(* Visualisation VISU_2_UDP
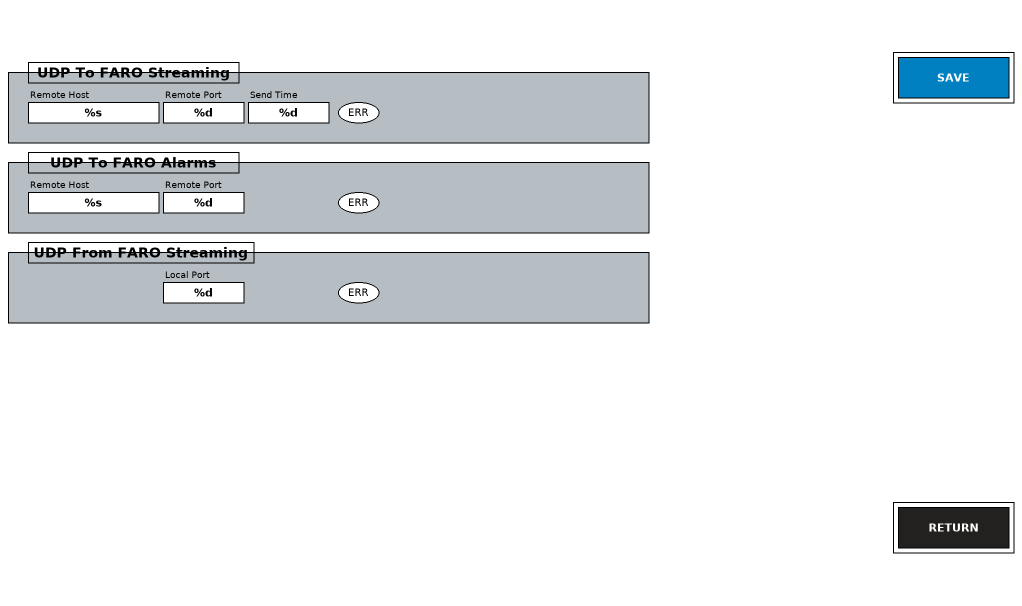
rounded rectangle at (905,505)-(1016,546): text "RETURN"; opens VISU_1_ALARMS
rectangle at (20,0)-(506,51): text "UDP STREAMING"
rectangle at (20,550)-(351,601): text "%s"; shows INPUTS.sVisuTime
rounded rectangle at (905,55)-(1016,96): text "SAVE"; alarm colour if PARAMS.Save; toggles PARAMS.Save
rectangle at (35,100)-(166,121): text "%s"; shows PARAMS.sUDPSendHost; editable
ellipse at (345,100)-(386,121): text "ERR"; alarm colour if TOFARO.fbUdpSend.bError
rectangle at (170,100)-(251,121): text "%d"; shows PARAMS.nUDPSendPort; editable
rectangle at (255,100)-(336,121): text "%d"; shows PARAMS.nUDPSendTime; editable 0..
rectangle at (35,85)-(126,101): text "Remote Host"
rectangle at (170,85)-(251,101): text "Remote Port"
rectangle at (255,85)-(336,101): text "Send Time"
rectangle at (35,60)-(246,81): text "UDP To FARO Streaming"
rectangle at (730,550)-(896,601): text "SAVED!"; invisible if PARAMS.Saved
ellipse at (345,280)-(386,301): text "ERR"; alarm colour if TOFARO.fbUdpRecv.bError
rectangle at (170,280)-(251,301): text "%d"; shows PARAMS.nUDPRecvPort; editable
rectangle at (170,265)-(251,281): text "Local Port"
rectangle at (35,240)-(261,261): text "UDP From FARO Streaming"
rectangle at (35,190)-(166,211): text "%s"; shows PARAMS.sUDPAlarmsHost; editable
ellipse at (345,190)-(386,211): text "ERR"; alarm colour if ALARMS.fbUdpSend.bError
rectangle at (170,190)-(251,211): text "%d"; shows PARAMS.nUDPAlarmsPort; editable
rectangle at (35,175)-(126,191): text "Remote Host"
rectangle at (170,175)-(251,191): text "Remote Port"
rectangle at (35,150)-(246,171): text "UDP To FARO Alarms"
5 more shapes without text or variables
*)

(* Visualisation VISU_CAL_CYLINDERS1
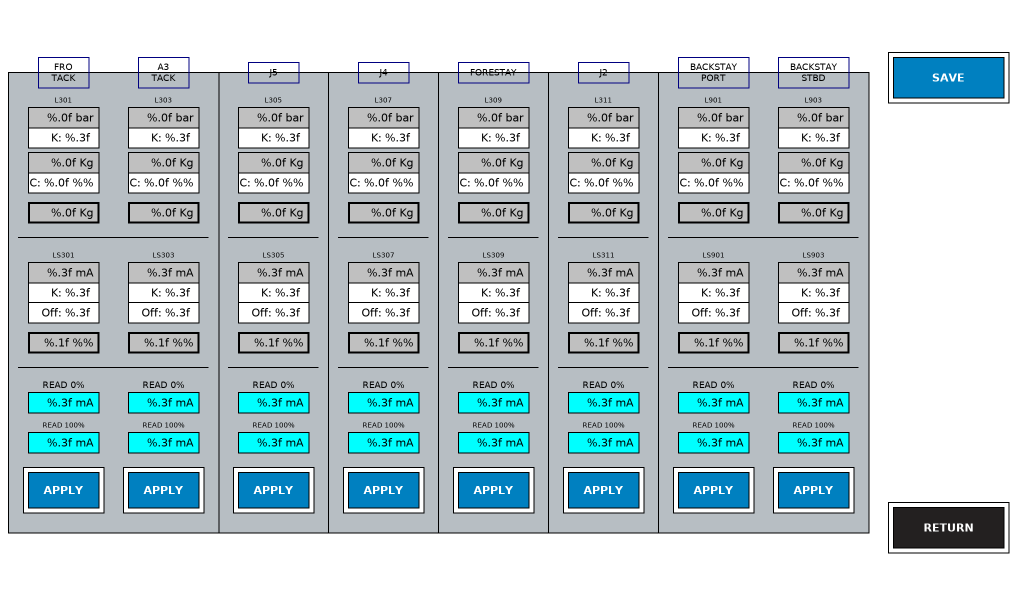
rectangle at (20,0)-(426,51): text "CAL: CYLINDERS 1"
rectangle at (20,550)-(331,601): text "%s"; shows INPUTS.sVisuTime
rounded rectangle at (905,55)-(1016,96): text "SAVE"; alarm colour if PARAMS.Save; toggles PARAMS.Save
rounded rectangle at (905,505)-(1016,546): text "RETURN"; opens VISU_1_CYLINDERS1
rectangle at (725,550)-(891,601): text "SAVED!"; invisible if PARAMS.Saved
rectangle at (40,245)-(111,261): text "LS301"
rectangle at (40,280)-(111,301): text "K: %.3f"; shows LS301.Cal_K; runs INTERN ASSIGN INPUTS.PresSelCalStbd[9]:=(FALSE); editable
rectangle at (40,260)-(111,281): text "%.3f mA"; shows LS301.Raw; alarm colour if LS301.Err; runs INTERN ASSIGN INPUTS.PresSelCalStbd[9]:=(FALSE)
rectangle at (40,300)-(111,321): text "Off: %.3f"; shows LS301.Cal_Off; runs INTERN ASSIGN INPUTS.PresSelCalStbd[9]:=(FALSE); editable
rectangle at (40,430)-(111,451): text "%.3f mA"; shows LS301.Cal_Max; alarm colour if LS301.Cal_Max = 0.0; runs INTERN ASSIGN INPUTS.PresSelCalStbd[9]:=(FALSE); editable
rectangle at (40,375)-(111,391): text "READ 0%"
rectangle at (40,415)-(111,431): text "READ 100%"
rounded rectangle at (40,470)-(111,506): text "APPLY"; toggles LS301.Cal_Apply
rectangle at (140,245)-(211,261): text "LS303"
rectangle at (140,280)-(211,301): text "K: %.3f"; shows LS303.Cal_K; runs INTERN ASSIGN INPUTS.PresSelCalStbd[9]:=(FALSE); editable
rectangle at (140,260)-(211,281): text "%.3f mA"; shows LS303.Raw; alarm colour if LS303.Err; runs INTERN ASSIGN INPUTS.PresSelCalStbd[9]:=(FALSE)
rectangle at (140,300)-(211,321): text "Off: %.3f"; shows LS303.Cal_Off; runs INTERN ASSIGN INPUTS.PresSelCalStbd[9]:=(FALSE); editable
rectangle at (140,430)-(211,451): text "%.3f mA"; shows LS303.Cal_Max; alarm colour if LS303.Cal_Max = 0.0; runs INTERN ASSIGN INPUTS.PresSelCalStbd[9]:=(FALSE); editable
rounded rectangle at (140,470)-(211,506): text "APPLY"; toggles LS303.Cal_Apply
rectangle at (690,280)-(761,301): text "K: %.3f"; shows LS901.Cal_K; runs INTERN ASSIGN INPUTS.PresSelCalStbd[9]:=(FALSE); editable
rectangle at (690,260)-(761,281): text "%.3f mA"; shows LS901.Raw; alarm colour if LS901.Err; runs INTERN ASSIGN INPUTS.PresSelCalStbd[9]:=(FALSE)
rectangle at (690,300)-(761,321): text "Off: %.3f"; shows LS901.Cal_Off; runs INTERN ASSIGN INPUTS.PresSelCalStbd[9]:=(FALSE); editable
rectangle at (690,390)-(761,411): text "%.3f mA"; shows LS901.Cal_Min; alarm colour if LS901.Cal_Min = 0.0; runs INTERN ASSIGN INPUTS.PresSelCalStbd[9]:=(FALSE); editable
rectangle at (690,430)-(761,451): text "%.3f mA"; shows LS901.Cal_Max; alarm colour if LS901.Cal_Max = 0.0; runs INTERN ASSIGN INPUTS.PresSelCalStbd[9]:=(FALSE); editable
rounded rectangle at (690,470)-(761,506): text "APPLY"; toggles LS901.Cal_Apply
rectangle at (790,280)-(861,301): text "K: %.3f"; shows LS903.Cal_K; runs INTERN ASSIGN INPUTS.PresSelCalStbd[9]:=(FALSE); editable
rectangle at (790,260)-(861,281): text "%.3f mA"; shows LS903.Raw; alarm colour if LS903.Err; runs INTERN ASSIGN INPUTS.PresSelCalStbd[9]:=(FALSE)
rectangle at (790,300)-(861,321): text "Off: %.3f"; shows LS903.Cal_Off; runs INTERN ASSIGN INPUTS.PresSelCalStbd[9]:=(FALSE); editable
rectangle at (790,390)-(861,411): text "%.3f mA"; shows LS903.Cal_Min; alarm colour if LS903.Cal_Min = 0.0; runs INTERN ASSIGN INPUTS.PresSelCalStbd[9]:=(FALSE); editable
rectangle at (790,430)-(861,451): text "%.3f mA"; shows LS903.Cal_Max; alarm colour if LS903.Cal_Max = 0.0; runs INTERN ASSIGN INPUTS.PresSelCalStbd[9]:=(FALSE); editable
rounded rectangle at (790,470)-(861,506): text "APPLY"; toggles LS903.Cal_Apply
rectangle at (580,280)-(651,301): text "K: %.3f"; shows LS311.Cal_K; runs INTERN ASSIGN INPUTS.PresSelCalStbd[9]:=(FALSE); editable
rectangle at (580,260)-(651,281): text "%.3f mA"; shows LS311.Raw; alarm colour if LS311.Err; runs INTERN ASSIGN INPUTS.PresSelCalStbd[9]:=(FALSE)
rectangle at (580,300)-(651,321): text "Off: %.3f"; shows LS311.Cal_Off; runs INTERN ASSIGN INPUTS.PresSelCalStbd[9]:=(FALSE); editable
rectangle at (580,390)-(651,411): text "%.3f mA"; shows LS311.Cal_Min; alarm colour if LS311.Cal_Min = 0.0; runs INTERN ASSIGN INPUTS.PresSelCalStbd[9]:=(FALSE); editable
rectangle at (580,430)-(651,451): text "%.3f mA"; shows LS311.Cal_Max; alarm colour if LS311.Cal_Max = 0.0; runs INTERN ASSIGN INPUTS.PresSelCalStbd[9]:=(FALSE); editable
rounded rectangle at (580,470)-(651,506): text "APPLY"; toggles LS311.Cal_Apply
rectangle at (250,280)-(321,301): text "K: %.3f"; shows LS305.Cal_K; runs INTERN ASSIGN INPUTS.PresSelCalStbd[9]:=(FALSE); editable
rectangle at (250,260)-(321,281): text "%.3f mA"; shows LS305.Raw; alarm colour if LS305.Err; runs INTERN ASSIGN INPUTS.PresSelCalStbd[9]:=(FALSE)
rectangle at (250,300)-(321,321): text "Off: %.3f"; shows LS305.Cal_Off; runs INTERN ASSIGN INPUTS.PresSelCalStbd[9]:=(FALSE); editable
rectangle at (250,390)-(321,411): text "%.3f mA"; shows LS305.Cal_Min; alarm colour if LS305.Cal_Min = 0.0; runs INTERN ASSIGN INPUTS.PresSelCalStbd[9]:=(FALSE); editable
rectangle at (250,430)-(321,451): text "%.3f mA"; shows LS305.Cal_Max; alarm colour if LS305.Cal_Max = 0.0; runs INTERN ASSIGN INPUTS.PresSelCalStbd[9]:=(FALSE); editable
rounded rectangle at (250,470)-(321,506): text "APPLY"; toggles LS305.Cal_Apply
rectangle at (360,280)-(431,301): text "K: %.3f"; shows LS307.Cal_K; runs INTERN ASSIGN INPUTS.PresSelCalStbd[9]:=(FALSE); editable
rectangle at (360,260)-(431,281): text "%.3f mA"; shows LS307.Raw; alarm colour if LS307.Err; runs INTERN ASSIGN INPUTS.PresSelCalStbd[9]:=(FALSE)
rectangle at (360,300)-(431,321): text "Off: %.3f"; shows LS307.Cal_Off; runs INTERN ASSIGN INPUTS.PresSelCalStbd[9]:=(FALSE); editable
rectangle at (360,390)-(431,411): text "%.3f mA"; shows LS307.Cal_Min; alarm colour if LS307.Cal_Min = 0.0; runs INTERN ASSIGN INPUTS.PresSelCalStbd[9]:=(FALSE); editable
rectangle at (360,430)-(431,451): text "%.3f mA"; shows LS307.Cal_Max; alarm colour if LS307.Cal_Max = 0.0; runs INTERN ASSIGN INPUTS.PresSelCalStbd[9]:=(FALSE); editable
rounded rectangle at (360,470)-(431,506): text "APPLY"; toggles LS307.Cal_Apply
rectangle at (40,390)-(111,411): text "%.3f mA"; shows LS301.Cal_Min; alarm colour if LS301.Cal_Min = 0.0; runs INTERN ASSIGN INPUTS.PresSelCalStbd[9]:=(FALSE); editable
rectangle at (140,390)-(211,411): text "%.3f mA"; shows LS303.Cal_Min; alarm colour if LS303.Cal_Min = 0.0; runs INTERN ASSIGN INPUTS.PresSelCalStbd[9]:=(FALSE); editable
rectangle at (40,90)-(111,106): text "L301"
rectangle at (40,200)-(111,221): text "%.0f Kg"; shows L301.Kg; runs INTERN ASSIGN INPUTS.PresSelCalStbd[9]:=(FALSE)
rectangle at (40,125)-(111,146): text "K: %.3f"; shows L301.Cal_K; runs INTERN ASSIGN INPUTS.PresSelCalStbd[9]:=(FALSE); editable
rectangle at (40,105)-(111,126): text "%.0f bar"; shows P301.Bar; alarm colour if P301.Err; runs INTERN ASSIGN INPUTS.PresSelCalStbd[9]:=(FALSE)
rectangle at (40,170)-(111,191): text "C: %.0f %%"; shows L301.Cal_C; runs INTERN ASSIGN INPUTS.PresSelCalStbd[9]:=(FALSE); editable
rectangle at (40,150)-(111,171): text "%.0f Kg"; shows L301.Raw; runs INTERN ASSIGN INPUTS.PresSelCalStbd[9]:=(FALSE)
rectangle at (40,330)-(111,351): text "%.1f %%"; shows LS301.Pos; runs INTERN ASSIGN INPUTS.PresSelCalStbd[9]:=(FALSE)
rectangle at (140,330)-(211,351): text "%.1f %%"; shows LS303.Pos; runs INTERN ASSIGN INPUTS.PresSelCalStbd[9]:=(FALSE)
rectangle at (690,330)-(761,351): text "%.1f %%"; shows LS901.Pos; runs INTERN ASSIGN INPUTS.PresSelCalStbd[9]:=(FALSE)
rectangle at (790,330)-(861,351): text "%.1f %%"; shows LS903.Pos; runs INTERN ASSIGN INPUTS.PresSelCalStbd[9]:=(FALSE)
rectangle at (580,330)-(651,351): text "%.1f %%"; shows LS311.Pos; runs INTERN ASSIGN INPUTS.PresSelCalStbd[9]:=(FALSE)
rectangle at (250,330)-(321,351): text "%.1f %%"; shows LS305.Pos; runs INTERN ASSIGN INPUTS.PresSelCalStbd[9]:=(FALSE)
rectangle at (360,330)-(431,351): text "%.1f %%"; shows LS307.Pos; runs INTERN ASSIGN INPUTS.PresSelCalStbd[9]:=(FALSE)
rectangle at (470,280)-(541,301): text "K: %.3f"; shows LS309.Cal_K; runs INTERN ASSIGN INPUTS.PresSelCalStbd[9]:=(FALSE); editable
rectangle at (470,260)-(541,281): text "%.3f mA"; shows LS309.Raw; alarm colour if LS309.Err; runs INTERN ASSIGN INPUTS.PresSelCalStbd[9]:=(FALSE)
rectangle at (470,300)-(541,321): text "Off: %.3f"; shows LS309.Cal_Off; runs INTERN ASSIGN INPUTS.PresSelCalStbd[9]:=(FALSE); editable
rectangle at (470,390)-(541,411): text "%.3f mA"; shows LS309.Cal_Min; alarm colour if LS309.Cal_Min = 0.0; runs INTERN ASSIGN INPUTS.PresSelCalStbd[9]:=(FALSE); editable
rectangle at (470,430)-(541,451): text "%.3f mA"; shows LS309.Cal_Max; alarm colour if LS309.Cal_Max = 0.0; runs INTERN ASSIGN INPUTS.PresSelCalStbd[9]:=(FALSE); editable
rounded rectangle at (470,470)-(541,506): text "APPLY"; toggles LS309.Cal_Apply
rectangle at (470,330)-(541,351): text "%.1f %%"; shows LS309.Pos; runs INTERN ASSIGN INPUTS.PresSelCalStbd[9]:=(FALSE)
rectangle at (140,90)-(211,106): text "L303"
rectangle at (140,200)-(211,221): text "%.0f Kg"; shows L303.Kg; runs INTERN ASSIGN INPUTS.PresSelCalStbd[9]:=(FALSE)
rectangle at (140,125)-(211,146): text "K: %.3f"; shows L303.Cal_K; runs INTERN ASSIGN INPUTS.PresSelCalStbd[9]:=(FALSE); editable
rectangle at (140,105)-(211,126): text "%.0f bar"; shows P303.Bar; alarm colour if P303.Err; runs INTERN ASSIGN INPUTS.PresSelCalStbd[9]:=(FALSE)
rectangle at (140,170)-(211,191): text "C: %.0f %%"; shows L303.Cal_C; runs INTERN ASSIGN INPUTS.PresSelCalStbd[9]:=(FALSE); editable
rectangle at (140,150)-(211,171): text "%.0f Kg"; shows L303.Raw; runs INTERN ASSIGN INPUTS.PresSelCalStbd[9]:=(FALSE)
rectangle at (250,90)-(321,106): text "L305"
rectangle at (250,200)-(321,221): text "%.0f Kg"; shows L305.Kg; runs INTERN ASSIGN INPUTS.PresSelCalStbd[9]:=(FALSE)
rectangle at (250,125)-(321,146): text "K: %.3f"; shows L305.Cal_K; runs INTERN ASSIGN INPUTS.PresSelCalStbd[9]:=(FALSE); editable
rectangle at (250,105)-(321,126): text "%.0f bar"; shows P305.Bar; alarm colour if P305.Err; runs INTERN ASSIGN INPUTS.PresSelCalStbd[9]:=(FALSE)
rectangle at (250,170)-(321,191): text "C: %.0f %%"; shows L305.Cal_C; runs INTERN ASSIGN INPUTS.PresSelCalStbd[9]:=(FALSE); editable
rectangle at (250,150)-(321,171): text "%.0f Kg"; shows L305.Raw; runs INTERN ASSIGN INPUTS.PresSelCalStbd[9]:=(FALSE)
rectangle at (250,245)-(321,261): text "LS305"
rectangle at (360,245)-(431,261): text "LS307"
rectangle at (470,245)-(541,261): text "LS309"
rectangle at (580,245)-(651,261): text "LS311"
rectangle at (690,245)-(761,261): text "LS901"
rectangle at (790,245)-(861,261): text "LS903"
rectangle at (360,90)-(431,106): text "L307"
rectangle at (360,200)-(431,221): text "%.0f Kg"; shows L307.Kg; runs INTERN ASSIGN INPUTS.PresSelCalStbd[9]:=(FALSE)
rectangle at (360,125)-(431,146): text "K: %.3f"; shows L307.Cal_K; runs INTERN ASSIGN INPUTS.PresSelCalStbd[9]:=(FALSE); editable
rectangle at (360,105)-(431,126): text "%.0f bar"; shows P307.Bar; alarm colour if P307.Err; runs INTERN ASSIGN INPUTS.PresSelCalStbd[9]:=(FALSE)
rectangle at (360,170)-(431,191): text "C: %.0f %%"; shows L307.Cal_C; runs INTERN ASSIGN INPUTS.PresSelCalStbd[9]:=(FALSE); editable
rectangle at (360,150)-(431,171): text "%.0f Kg"; shows L307.Raw; runs INTERN ASSIGN INPUTS.PresSelCalStbd[9]:=(FALSE)
rectangle at (470,90)-(541,106): text "L309"
rectangle at (470,200)-(541,221): text "%.0f Kg"; shows L309.Kg; runs INTERN ASSIGN INPUTS.PresSelCalStbd[9]:=(FALSE)
rectangle at (470,125)-(541,146): text "K: %.3f"; shows L309.Cal_K; runs INTERN ASSIGN INPUTS.PresSelCalStbd[9]:=(FALSE); editable
rectangle at (470,105)-(541,126): text "%.0f bar"; shows P309.Bar; alarm colour if P309.Err; runs INTERN ASSIGN INPUTS.PresSelCalStbd[9]:=(FALSE)
rectangle at (470,170)-(541,191): text "C: %.0f %%"; shows L309.Cal_C; runs INTERN ASSIGN INPUTS.PresSelCalStbd[9]:=(FALSE); editable
rectangle at (470,150)-(541,171): text "%.0f Kg"; shows L309.Raw; runs INTERN ASSIGN INPUTS.PresSelCalStbd[9]:=(FALSE)
rectangle at (580,90)-(651,106): text "L311"
rectangle at (580,200)-(651,221): text "%.0f Kg"; shows L311.Kg; runs INTERN ASSIGN INPUTS.PresSelCalStbd[9]:=(FALSE)
rectangle at (580,125)-(651,146): text "K: %.3f"; shows L311.Cal_K; runs INTERN ASSIGN INPUTS.PresSelCalStbd[9]:=(FALSE); editable
rectangle at (580,105)-(651,126): text "%.0f bar"; shows P311.Bar; alarm colour if P311.Err; runs INTERN ASSIGN INPUTS.PresSelCalStbd[9]:=(FALSE)
rectangle at (580,170)-(651,191): text "C: %.0f %%"; shows L311.Cal_C; runs INTERN ASSIGN INPUTS.PresSelCalStbd[9]:=(FALSE); editable
rectangle at (580,150)-(651,171): text "%.0f Kg"; shows L311.Raw; runs INTERN ASSIGN INPUTS.PresSelCalStbd[9]:=(FALSE)
rectangle at (690,90)-(761,106): text "L901"
rectangle at (690,200)-(761,221): text "%.0f Kg"; shows L901.Kg; runs INTERN ASSIGN INPUTS.PresSelCalStbd[9]:=(FALSE)
rectangle at (690,125)-(761,146): text "K: %.3f"; shows L901.Cal_K; runs INTERN ASSIGN INPUTS.PresSelCalStbd[9]:=(FALSE); editable
rectangle at (690,105)-(761,126): text "%.0f bar"; shows P901.Bar; alarm colour if P901.Err; runs INTERN ASSIGN INPUTS.PresSelCalStbd[9]:=(FALSE)
rectangle at (690,170)-(761,191): text "C: %.0f %%"; shows L901.Cal_C; runs INTERN ASSIGN INPUTS.PresSelCalStbd[9]:=(FALSE); editable
rectangle at (690,150)-(761,171): text "%.0f Kg"; shows L901.Raw; runs INTERN ASSIGN INPUTS.PresSelCalStbd[9]:=(FALSE)
rectangle at (790,90)-(861,106): text "L903"
rectangle at (790,200)-(861,221): text "%.0f Kg"; shows L903.Kg; runs INTERN ASSIGN INPUTS.PresSelCalStbd[9]:=(FALSE)
rectangle at (790,125)-(861,146): text "K: %.3f"; shows L903.Cal_K; runs INTERN ASSIGN INPUTS.PresSelCalStbd[9]:=(FALSE); editable
rectangle at (790,105)-(861,126): text "%.0f bar"; shows P903.Bar; alarm colour if P903.Err; runs INTERN ASSIGN INPUTS.PresSelCalStbd[9]:=(FALSE)
rectangle at (790,170)-(861,191): text "C: %.0f %%"; shows L903.Cal_C; runs INTERN ASSIGN INPUTS.PresSelCalStbd[9]:=(FALSE); editable
rectangle at (790,150)-(861,171): text "%.0f Kg"; shows L903.Raw; runs INTERN ASSIGN INPUTS.PresSelCalStbd[9]:=(FALSE)
rectangle at (260,60)-(311,81): text "J5"
rectangle at (370,60)-(421,81): text "J4"
rectangle at (470,60)-(541,81): text "FORESTAY"
rectangle at (590,60)-(641,81): text "J2"
rectangle at (690,55)-(761,86): text "BACKSTAY / PORT"
rectangle at (790,55)-(861,86): text "BACKSTAY / STBD"
rectangle at (150,55)-(201,86): text "A3 / TACK"
rectangle at (50,55)-(101,86): text "FRO / TACK"
rectangle at (140,375)-(211,391): text "READ 0%"
rectangle at (140,415)-(211,431): text "READ 100%"
rectangle at (250,375)-(321,391): text "READ 0%"
rectangle at (250,415)-(321,431): text "READ 100%"
rectangle at (360,375)-(431,391): text "READ 0%"
rectangle at (360,415)-(431,431): text "READ 100%"
rectangle at (470,375)-(541,391): text "READ 0%"
rectangle at (470,415)-(541,431): text "READ 100%"
rectangle at (580,375)-(651,391): text "READ 0%"
rectangle at (580,415)-(651,431): text "READ 100%"
rectangle at (690,375)-(761,391): text "READ 0%"
rectangle at (690,415)-(761,431): text "READ 100%"
rectangle at (790,375)-(861,391): text "READ 0%"
rectangle at (790,415)-(861,431): text "READ 100%"
28 more shapes without text or variables
*)

(* Visualisation VISU_CAL_CYLINDERS2
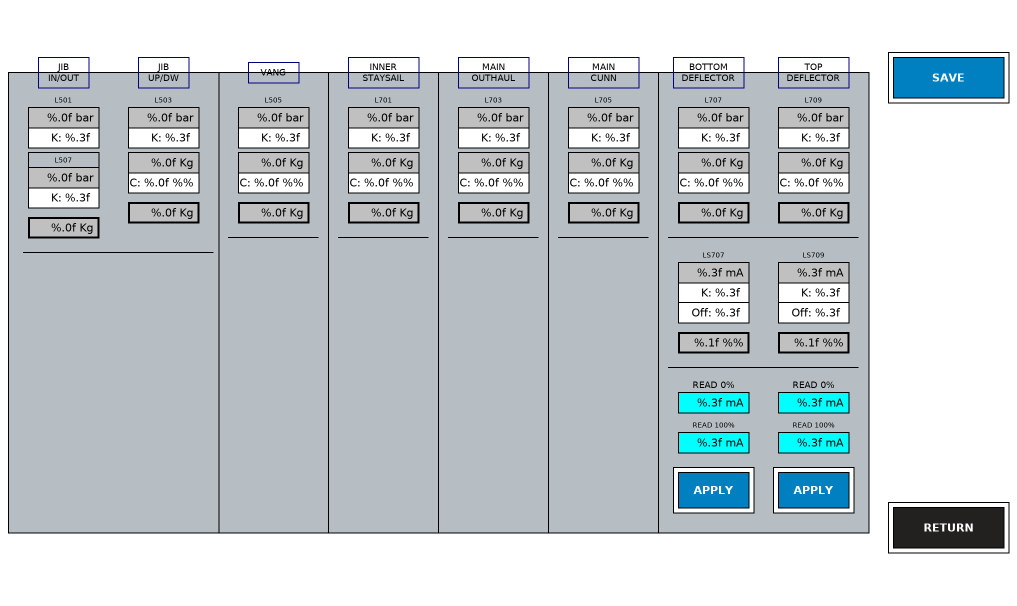
rectangle at (20,0)-(426,51): text "CAL: CYLINDERS 2"
rectangle at (20,550)-(331,601): text "%s"; shows INPUTS.sVisuTime
rounded rectangle at (905,55)-(1016,96): text "SAVE"; alarm colour if PARAMS.Save; toggles PARAMS.Save
rounded rectangle at (905,505)-(1016,546): text "RETURN"; opens VISU_1_CYLINDERS2
rectangle at (730,550)-(896,601): text "SAVED!"; invisible if PARAMS.Saved
rectangle at (690,245)-(761,261): text "LS707"
rectangle at (690,280)-(761,301): text "K: %.3f"; shows LS707.Cal_K; runs INTERN ASSIGN INPUTS.PresSelCalStbd[9]:=(FALSE); editable
rectangle at (690,260)-(761,281): text "%.3f mA"; shows LS707.Raw; alarm colour if LS707.Err; runs INTERN ASSIGN INPUTS.PresSelCalStbd[9]:=(FALSE)
rectangle at (690,300)-(761,321): text "Off: %.3f"; shows LS707.Cal_Off; runs INTERN ASSIGN INPUTS.PresSelCalStbd[9]:=(FALSE); editable
rectangle at (690,430)-(761,451): text "%.3f mA"; shows LS707.Cal_Max; alarm colour if LS707.Cal_Max = 0.0; runs INTERN ASSIGN INPUTS.PresSelCalStbd[9]:=(FALSE); editable
rectangle at (690,375)-(761,391): text "READ 0%"
rectangle at (690,415)-(761,431): text "READ 100%"
rounded rectangle at (690,470)-(761,506): text "APPLY"; toggles LS707.Cal_Apply
rectangle at (790,245)-(861,261): text "LS709"
rectangle at (790,280)-(861,301): text "K: %.3f"; shows LS709.Cal_K; runs INTERN ASSIGN INPUTS.PresSelCalStbd[9]:=(FALSE); editable
rectangle at (790,260)-(861,281): text "%.3f mA"; shows LS709.Raw; alarm colour if LS709.Err; runs INTERN ASSIGN INPUTS.PresSelCalStbd[9]:=(FALSE)
rectangle at (790,300)-(861,321): text "Off: %.3f"; shows LS709.Cal_Off; runs INTERN ASSIGN INPUTS.PresSelCalStbd[9]:=(FALSE); editable
rectangle at (790,430)-(861,451): text "%.3f mA"; shows LS709.Cal_Max; alarm colour if LS709.Cal_Max = 0.0; runs INTERN ASSIGN INPUTS.PresSelCalStbd[9]:=(FALSE); editable
rectangle at (790,375)-(861,391): text "READ 0%"
rectangle at (790,415)-(861,431): text "READ 100%"
rounded rectangle at (790,470)-(861,506): text "APPLY"; toggles LS709.Cal_Apply
rectangle at (690,390)-(761,411): text "%.3f mA"; shows LS707.Cal_Min; alarm colour if LS707.Cal_Min = 0.0; runs INTERN ASSIGN INPUTS.PresSelCalStbd[9]:=(FALSE); editable
rectangle at (790,390)-(861,411): text "%.3f mA"; shows LS709.Cal_Min; alarm colour if LS709.Cal_Min = 0.0; runs INTERN ASSIGN INPUTS.PresSelCalStbd[9]:=(FALSE); editable
rectangle at (690,330)-(761,351): text "%.1f %%"; shows LS707.Pos; runs INTERN ASSIGN INPUTS.PresSelCalStbd[9]:=(FALSE)
rectangle at (790,330)-(861,351): text "%.1f %%"; shows LS709.Pos; runs INTERN ASSIGN INPUTS.PresSelCalStbd[9]:=(FALSE)
rectangle at (40,90)-(111,106): text "L501"
rectangle at (40,215)-(111,236): text "%.0f Kg"; shows L501_7; runs INTERN ASSIGN INPUTS.PresSelCalStbd[9]:=(FALSE)
rectangle at (40,125)-(111,146): text "K: %.3f"; shows L501.Cal_K; runs INTERN ASSIGN INPUTS.PresSelCalStbd[9]:=(FALSE); editable
rectangle at (40,105)-(111,126): text "%.0f bar"; shows P501.Bar; alarm colour if P501.Err; runs INTERN ASSIGN INPUTS.PresSelCalStbd[9]:=(FALSE)
rectangle at (140,90)-(211,106): text "L503"
rectangle at (140,200)-(211,221): text "%.0f Kg"; shows L503.Kg; runs INTERN ASSIGN INPUTS.PresSelCalStbd[9]:=(FALSE)
rectangle at (140,125)-(211,146): text "K: %.3f"; shows L503.Cal_K; runs INTERN ASSIGN INPUTS.PresSelCalStbd[9]:=(FALSE); editable
rectangle at (140,105)-(211,126): text "%.0f bar"; shows P503.Bar; alarm colour if P503.Err; runs INTERN ASSIGN INPUTS.PresSelCalStbd[9]:=(FALSE)
rectangle at (140,170)-(211,191): text "C: %.0f %%"; shows L503.Cal_C; runs INTERN ASSIGN INPUTS.PresSelCalStbd[9]:=(FALSE); editable
rectangle at (140,150)-(211,171): text "%.0f Kg"; shows L503.Raw; runs INTERN ASSIGN INPUTS.PresSelCalStbd[9]:=(FALSE)
rectangle at (690,90)-(761,106): text "L707"
rectangle at (690,200)-(761,221): text "%.0f Kg"; shows L707.Kg; runs INTERN ASSIGN INPUTS.PresSelCalStbd[9]:=(FALSE)
rectangle at (690,125)-(761,146): text "K: %.3f"; shows L707.Cal_K; runs INTERN ASSIGN INPUTS.PresSelCalStbd[9]:=(FALSE); editable
rectangle at (690,105)-(761,126): text "%.0f bar"; shows P707.Bar; alarm colour if P707.Err; runs INTERN ASSIGN INPUTS.PresSelCalStbd[9]:=(FALSE)
rectangle at (690,170)-(761,191): text "C: %.0f %%"; shows L707.Cal_C; runs INTERN ASSIGN INPUTS.PresSelCalStbd[9]:=(FALSE); editable
rectangle at (690,150)-(761,171): text "%.0f Kg"; shows L707.Raw; runs INTERN ASSIGN INPUTS.PresSelCalStbd[9]:=(FALSE)
rectangle at (790,90)-(861,106): text "L709"
rectangle at (790,200)-(861,221): text "%.0f Kg"; shows L709.Kg; runs INTERN ASSIGN INPUTS.PresSelCalStbd[9]:=(FALSE)
rectangle at (790,125)-(861,146): text "K: %.3f"; shows L709.Cal_K; runs INTERN ASSIGN INPUTS.PresSelCalStbd[9]:=(FALSE); editable
rectangle at (790,105)-(861,126): text "%.0f bar"; shows P709.Bar; alarm colour if P709.Err; runs INTERN ASSIGN INPUTS.PresSelCalStbd[9]:=(FALSE)
rectangle at (790,170)-(861,191): text "C: %.0f %%"; shows L709.Cal_C; runs INTERN ASSIGN INPUTS.PresSelCalStbd[9]:=(FALSE); editable
rectangle at (790,150)-(861,171): text "%.0f Kg"; shows L709.Raw; runs INTERN ASSIGN INPUTS.PresSelCalStbd[9]:=(FALSE)
rectangle at (250,90)-(321,106): text "L505"
rectangle at (250,200)-(321,221): text "%.0f Kg"; shows L505.Kg; runs INTERN ASSIGN INPUTS.PresSelCalStbd[9]:=(FALSE)
rectangle at (250,125)-(321,146): text "K: %.3f"; shows L505.Cal_K; runs INTERN ASSIGN INPUTS.PresSelCalStbd[9]:=(FALSE); editable
rectangle at (250,105)-(321,126): text "%.0f bar"; shows P505.Bar; alarm colour if P505.Err; runs INTERN ASSIGN INPUTS.PresSelCalStbd[9]:=(FALSE)
rectangle at (250,170)-(321,191): text "C: %.0f %%"; shows L505.Cal_C; runs INTERN ASSIGN INPUTS.PresSelCalStbd[9]:=(FALSE); editable
rectangle at (250,150)-(321,171): text "%.0f Kg"; shows L505.Raw; runs INTERN ASSIGN INPUTS.PresSelCalStbd[9]:=(FALSE)
rectangle at (360,90)-(431,106): text "L701"
rectangle at (360,200)-(431,221): text "%.0f Kg"; shows L701.Kg; runs INTERN ASSIGN INPUTS.PresSelCalStbd[9]:=(FALSE)
rectangle at (360,125)-(431,146): text "K: %.3f"; shows L701.Cal_K; runs INTERN ASSIGN INPUTS.PresSelCalStbd[9]:=(FALSE); editable
rectangle at (360,105)-(431,126): text "%.0f bar"; shows P701.Bar; alarm colour if P701.Err; runs INTERN ASSIGN INPUTS.PresSelCalStbd[9]:=(FALSE)
rectangle at (360,170)-(431,191): text "C: %.0f %%"; shows L701.Cal_C; runs INTERN ASSIGN INPUTS.PresSelCalStbd[9]:=(FALSE); editable
rectangle at (360,150)-(431,171): text "%.0f Kg"; shows L701.Raw; runs INTERN ASSIGN INPUTS.PresSelCalStbd[9]:=(FALSE)
rectangle at (470,90)-(541,106): text "L703"
rectangle at (470,200)-(541,221): text "%.0f Kg"; shows L703.Kg; runs INTERN ASSIGN INPUTS.PresSelCalStbd[9]:=(FALSE)
rectangle at (470,125)-(541,146): text "K: %.3f"; shows L703.Cal_K; runs INTERN ASSIGN INPUTS.PresSelCalStbd[9]:=(FALSE); editable
rectangle at (470,105)-(541,126): text "%.0f bar"; shows P703.Bar; alarm colour if P703.Err; runs INTERN ASSIGN INPUTS.PresSelCalStbd[9]:=(FALSE)
rectangle at (470,170)-(541,191): text "C: %.0f %%"; shows L703.Cal_C; runs INTERN ASSIGN INPUTS.PresSelCalStbd[9]:=(FALSE); editable
rectangle at (470,150)-(541,171): text "%.0f Kg"; shows L703.Raw; runs INTERN ASSIGN INPUTS.PresSelCalStbd[9]:=(FALSE)
rectangle at (580,90)-(651,106): text "L705"
rectangle at (580,200)-(651,221): text "%.0f Kg"; shows L705.Kg; runs INTERN ASSIGN INPUTS.PresSelCalStbd[9]:=(FALSE)
rectangle at (580,125)-(651,146): text "K: %.3f"; shows L705.Cal_K; runs INTERN ASSIGN INPUTS.PresSelCalStbd[9]:=(FALSE); editable
rectangle at (580,105)-(651,126): text "%.0f bar"; shows P705.Bar; alarm colour if P705.Err; runs INTERN ASSIGN INPUTS.PresSelCalStbd[9]:=(FALSE)
rectangle at (580,170)-(651,191): text "C: %.0f %%"; shows L705.Cal_C; runs INTERN ASSIGN INPUTS.PresSelCalStbd[9]:=(FALSE); editable
rectangle at (580,150)-(651,171): text "%.0f Kg"; shows L705.Raw; runs INTERN ASSIGN INPUTS.PresSelCalStbd[9]:=(FALSE)
rectangle at (40,150)-(111,166): text "L507"
rectangle at (40,185)-(111,206): text "K: %.3f"; shows L501.Cal_C; runs INTERN ASSIGN INPUTS.PresSelCalStbd[9]:=(FALSE); editable
rectangle at (40,165)-(111,186): text "%.0f bar"; shows P507.Bar; alarm colour if P507.Err; runs INTERN ASSIGN INPUTS.PresSelCalStbd[9]:=(FALSE)
rectangle at (260,60)-(311,81): text "VANG"
rectangle at (50,55)-(101,86): text "JIB / IN/OUT"
rectangle at (150,55)-(201,86): text "JIB / UP/DW"
rectangle at (685,55)-(756,86): text "BOTTOM / DEFLECTOR"
rectangle at (790,55)-(861,86): text "TOP / DEFLECTOR"
rectangle at (360,55)-(431,86): text "INNER / STAYSAIL"
rectangle at (470,55)-(541,86): text "MAIN / OUTHAUL"
rectangle at (580,55)-(651,86): text "MAIN / CUNN"
17 more shapes without text or variables
*)

(* Visualisation VISU_CAL_SPECIAL
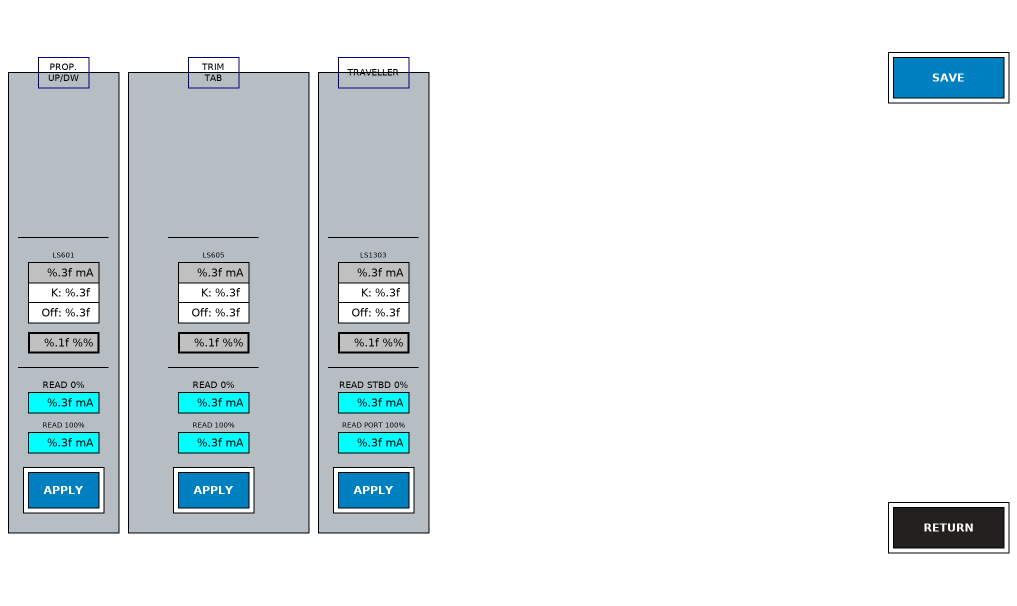
rectangle at (20,0)-(426,51): text "CAL: SPECIAL"
rectangle at (20,550)-(331,601): text "%s"; shows INPUTS.sVisuTime
rounded rectangle at (905,55)-(1016,96): text "SAVE"; alarm colour if PARAMS.Save; toggles PARAMS.Save
rounded rectangle at (905,505)-(1016,546): text "RETURN"; opens VISU_1_SPECIAL
rectangle at (730,550)-(896,601): text "SAVED!"; invisible if PARAMS.Saved
rectangle at (190,245)-(261,261): text "LS605"
rectangle at (190,330)-(261,351): text "%.1f %%"; shows LS605.Pos; runs INTERN ASSIGN INPUTS.PresSelCalStbd[9]:=(FALSE)
rectangle at (190,280)-(261,301): text "K: %.3f"; shows LS605.Cal_K; runs INTERN ASSIGN INPUTS.PresSelCalStbd[9]:=(FALSE); editable
rectangle at (190,260)-(261,281): text "%.3f mA"; shows LS605.Raw; alarm colour if LS605.Err; runs INTERN ASSIGN INPUTS.PresSelCalStbd[9]:=(FALSE)
rectangle at (190,300)-(261,321): text "Off: %.3f"; shows LS605.Cal_Off; runs INTERN ASSIGN INPUTS.PresSelCalStbd[9]:=(FALSE); editable
rectangle at (190,390)-(261,411): text "%.3f mA"; shows LS605.Cal_Min; alarm colour if LS605.Cal_Min = 0.0; runs INTERN ASSIGN INPUTS.PresSelCalStbd[9]:=(FALSE); editable
rectangle at (190,430)-(261,451): text "%.3f mA"; shows LS605.Cal_Max; alarm colour if LS605.Cal_Max = 0.0; runs INTERN ASSIGN INPUTS.PresSelCalStbd[9]:=(FALSE); editable
rectangle at (190,375)-(261,391): text "READ 0%"
rectangle at (190,415)-(261,431): text "READ 100%"
rounded rectangle at (190,470)-(261,506): text "APPLY"; toggles LS605.Cal_Apply
rectangle at (200,55)-(251,86): text "TRIM / TAB"
rectangle at (40,245)-(111,261): text "LS601"
rectangle at (40,330)-(111,351): text "%.1f %%"; shows LS601.Pos; runs INTERN ASSIGN INPUTS.PresSelCalStbd[9]:=(FALSE)
rectangle at (40,280)-(111,301): text "K: %.3f"; shows LS601.Cal_K; runs INTERN ASSIGN INPUTS.PresSelCalStbd[9]:=(FALSE); editable
rectangle at (40,260)-(111,281): text "%.3f mA"; shows LS601.Raw; alarm colour if LS601.Err; runs INTERN ASSIGN INPUTS.PresSelCalStbd[9]:=(FALSE)
rectangle at (40,300)-(111,321): text "Off: %.3f"; shows LS601.Cal_Off; runs INTERN ASSIGN INPUTS.PresSelCalStbd[9]:=(FALSE); editable
rectangle at (40,390)-(111,411): text "%.3f mA"; shows LS601.Cal_Min; alarm colour if LS601.Cal_Min = 0.0; runs INTERN ASSIGN INPUTS.PresSelCalStbd[9]:=(FALSE); editable
rectangle at (40,430)-(111,451): text "%.3f mA"; shows LS601.Cal_Max; alarm colour if LS601.Cal_Max = 0.0; runs INTERN ASSIGN INPUTS.PresSelCalStbd[9]:=(FALSE); editable
rectangle at (40,375)-(111,391): text "READ 0%"
rectangle at (40,415)-(111,431): text "READ 100%"
rounded rectangle at (40,470)-(111,506): text "APPLY"; toggles LS601.Cal_Apply
rectangle at (50,55)-(101,86): text "PROP. / UP/DW"
rectangle at (350,245)-(421,261): text "LS1303"
rectangle at (350,330)-(421,351): text "%.1f %%"; shows LS1303.Pos; runs INTERN ASSIGN INPUTS.PresSelCalStbd[9]:=(FALSE)
rectangle at (350,280)-(421,301): text "K: %.3f"; shows LS1303.Cal_K; runs INTERN ASSIGN INPUTS.PresSelCalStbd[9]:=(FALSE); editable
rectangle at (350,260)-(421,281): text "%.3f mA"; shows LS1303.Raw; alarm colour if LS1303.Err; runs INTERN ASSIGN INPUTS.PresSelCalStbd[9]:=(FALSE)
rectangle at (350,300)-(421,321): text "Off: %.3f"; shows LS1303.Cal_Off; runs INTERN ASSIGN INPUTS.PresSelCalStbd[9]:=(FALSE); editable
rectangle at (350,390)-(421,411): text "%.3f mA"; shows LS1303.Cal_Min; alarm colour if LS1303.Cal_Min = 0.0; runs INTERN ASSIGN INPUTS.PresSelCalStbd[9]:=(FALSE); editable
rectangle at (350,430)-(421,451): text "%.3f mA"; shows LS1303.Cal_Max; alarm colour if LS1303.Cal_Max = 0.0; runs INTERN ASSIGN INPUTS.PresSelCalStbd[9]:=(FALSE); editable
rectangle at (335,375)-(436,391): text "READ STBD 0%"
rectangle at (335,415)-(436,431): text "READ PORT 100%"
rounded rectangle at (350,470)-(421,506): text "APPLY"; toggles LS1303.Cal_Apply
rectangle at (350,55)-(421,86): text "TRAVELLER"
14 more shapes without text or variables
*)

(* Visualisation VISU_CAL_WB
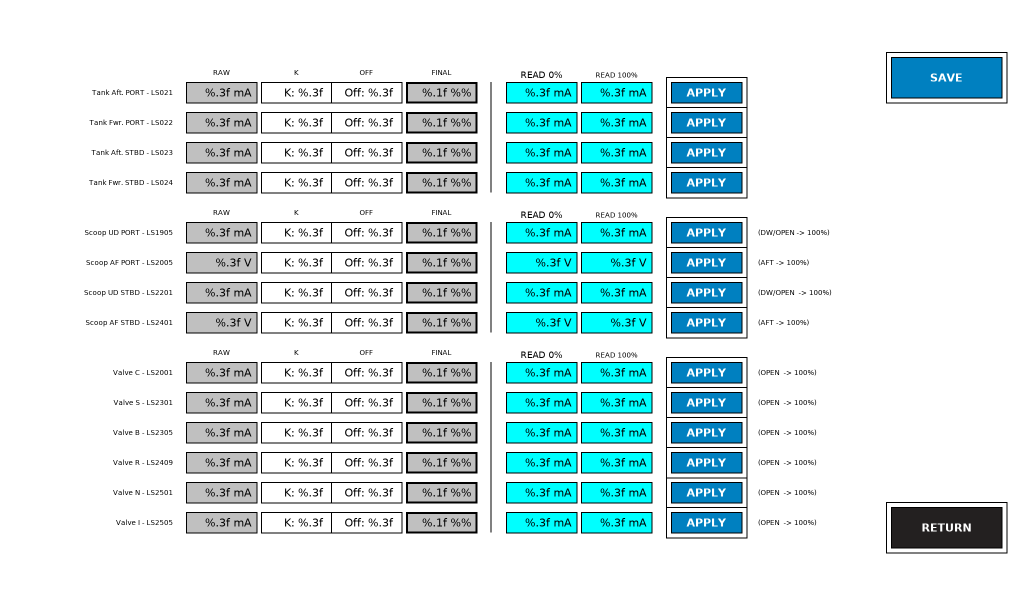
rectangle at (200,340)-(271,361): text "RAW"
rectangle at (420,340)-(491,361): text "FINAL"
rectangle at (275,340)-(346,361): text "K"
rectangle at (345,340)-(416,361): text "OFF"
rectangle at (200,200)-(271,221): text "RAW"
rectangle at (420,200)-(491,221): text "FINAL"
rectangle at (275,200)-(346,221): text "K"
rectangle at (345,200)-(416,221): text "OFF"
rectangle at (200,60)-(271,81): text "RAW"
rectangle at (420,60)-(491,81): text "FINAL"
rectangle at (275,60)-(346,81): text "K"
rectangle at (345,60)-(416,81): text "OFF"
rectangle at (20,0)-(426,51): text "CAL: WATER BALLAST"
rectangle at (20,550)-(331,601): text "%s"; shows INPUTS.sVisuTime
rounded rectangle at (905,55)-(1016,96): text "SAVE"; alarm colour if PARAMS.Save; toggles PARAMS.Save
rounded rectangle at (905,505)-(1016,546): text "RETURN"; opens VISU_1_WB
rectangle at (730,550)-(896,601): text "SAVED!"; invisible if PARAMS.Saved
rectangle at (45,80)-(191,101): text "Tank Aft. PORT - LS021"
rectangle at (275,80)-(346,101): text "K: %.3f"; shows LS021.Cal_K; runs INTERN ASSIGN INPUTS.PresSelCalStbd[9]:=(FALSE); editable
rectangle at (200,80)-(271,101): text "%.3f mA"; shows LS021.Raw; alarm colour if LS021.Err; runs INTERN ASSIGN INPUTS.PresSelCalStbd[9]:=(FALSE)
rectangle at (345,80)-(416,101): text "Off: %.3f"; shows LS021.Cal_Off; runs INTERN ASSIGN INPUTS.PresSelCalStbd[9]:=(FALSE); editable
rectangle at (595,80)-(666,101): text "%.3f mA"; shows LS021.Cal_Max; alarm colour if LS021.Cal_Max = 0.0; runs INTERN ASSIGN INPUTS.PresSelCalStbd[9]:=(FALSE); editable
rectangle at (520,65)-(591,81): text "READ 0%"
rectangle at (595,65)-(666,81): text "READ 100%"
rounded rectangle at (685,80)-(756,101): text "APPLY"; toggles LS021.Cal_Apply
rectangle at (520,80)-(591,101): text "%.3f mA"; shows LS021.Cal_Min; alarm colour if LS021.Cal_Min = 0.0; runs INTERN ASSIGN INPUTS.PresSelCalStbd[9]:=(FALSE); editable
rectangle at (420,80)-(491,101): text "%.1f %%"; shows LS021.Pos; runs INTERN ASSIGN INPUTS.PresSelCalStbd[9]:=(FALSE)
rectangle at (45,110)-(191,131): text "Tank Fwr. PORT - LS022"
rectangle at (275,110)-(346,131): text "K: %.3f"; shows LS022.Cal_K; runs INTERN ASSIGN INPUTS.PresSelCalStbd[9]:=(FALSE); editable
rectangle at (200,110)-(271,131): text "%.3f mA"; shows LS022.Raw; alarm colour if LS022.Err; runs INTERN ASSIGN INPUTS.PresSelCalStbd[9]:=(FALSE)
rectangle at (345,110)-(416,131): text "Off: %.3f"; shows LS022.Cal_Off; runs INTERN ASSIGN INPUTS.PresSelCalStbd[9]:=(FALSE); editable
rectangle at (595,110)-(666,131): text "%.3f mA"; shows LS022.Cal_Max; alarm colour if LS022.Cal_Max = 0.0; runs INTERN ASSIGN INPUTS.PresSelCalStbd[9]:=(FALSE); editable
rounded rectangle at (685,110)-(756,131): text "APPLY"; toggles LS022.Cal_Apply
rectangle at (520,110)-(591,131): text "%.3f mA"; shows LS022.Cal_Min; alarm colour if LS022.Cal_Min = 0.0; runs INTERN ASSIGN INPUTS.PresSelCalStbd[9]:=(FALSE); editable
rectangle at (420,110)-(491,131): text "%.1f %%"; shows LS022.Pos; runs INTERN ASSIGN INPUTS.PresSelCalStbd[9]:=(FALSE)
rounded rectangle at (685,140)-(756,161): text "APPLY"; toggles LS023.Cal_Apply
rounded rectangle at (685,170)-(756,191): text "APPLY"; toggles LS024.Cal_Apply
rectangle at (595,140)-(666,161): text "%.3f mA"; shows LS023.Cal_Max; alarm colour if LS023.Cal_Max = 0.0; runs INTERN ASSIGN INPUTS.PresSelCalStbd[9]:=(FALSE); editable
rectangle at (520,140)-(591,161): text "%.3f mA"; shows LS023.Cal_Min; alarm colour if LS023.Cal_Min = 0.0; runs INTERN ASSIGN INPUTS.PresSelCalStbd[9]:=(FALSE); editable
rectangle at (595,170)-(666,191): text "%.3f mA"; shows LS024.Cal_Max; alarm colour if LS024.Cal_Max = 0.0; runs INTERN ASSIGN INPUTS.PresSelCalStbd[9]:=(FALSE); editable
rectangle at (520,170)-(591,191): text "%.3f mA"; shows LS024.Cal_Min; alarm colour if LS024.Cal_Min = 0.0; runs INTERN ASSIGN INPUTS.PresSelCalStbd[9]:=(FALSE); editable
rectangle at (45,140)-(191,161): text "Tank Aft. STBD - LS023"
rectangle at (275,140)-(346,161): text "K: %.3f"; shows LS023.Cal_K; runs INTERN ASSIGN INPUTS.PresSelCalStbd[9]:=(FALSE); editable
rectangle at (200,140)-(271,161): text "%.3f mA"; shows LS023.Raw; alarm colour if LS023.Err; runs INTERN ASSIGN INPUTS.PresSelCalStbd[9]:=(FALSE)
rectangle at (345,140)-(416,161): text "Off: %.3f"; shows LS023.Cal_Off; runs INTERN ASSIGN INPUTS.PresSelCalStbd[9]:=(FALSE); editable
rectangle at (420,140)-(491,161): text "%.1f %%"; shows LS023.Pos; runs INTERN ASSIGN INPUTS.PresSelCalStbd[9]:=(FALSE)
rectangle at (45,170)-(191,191): text "Tank Fwr. STBD - LS024"
rectangle at (275,170)-(346,191): text "K: %.3f"; shows LS024.Cal_K; runs INTERN ASSIGN INPUTS.PresSelCalStbd[9]:=(FALSE); editable
rectangle at (200,170)-(271,191): text "%.3f mA"; shows LS024.Raw; alarm colour if LS024.Err; runs INTERN ASSIGN INPUTS.PresSelCalStbd[9]:=(FALSE)
rectangle at (345,170)-(416,191): text "Off: %.3f"; shows LS024.Cal_Off; runs INTERN ASSIGN INPUTS.PresSelCalStbd[9]:=(FALSE); editable
rectangle at (420,170)-(491,191): text "%.1f %%"; shows LS024.Pos; runs INTERN ASSIGN INPUTS.PresSelCalStbd[9]:=(FALSE)
rounded rectangle at (685,220)-(756,241): text "APPLY"; toggles LS1905.Cal_Apply
rectangle at (595,220)-(666,241): text "%.3f mA"; shows LS1905.Cal_Max; alarm colour if LS1905.Cal_Max = 0.0; runs INTERN ASSIGN INPUTS.PresSelCalStbd[9]:=(FALSE); editable
rectangle at (520,220)-(591,241): text "%.3f mA"; shows LS1905.Cal_Min; alarm colour if LS1905.Cal_Min = 0.0; runs INTERN ASSIGN INPUTS.PresSelCalStbd[9]:=(FALSE); editable
rectangle at (45,220)-(191,241): text "Scoop UD PORT - LS1905"
rectangle at (275,220)-(346,241): text "K: %.3f"; shows LS1905.Cal_K; runs INTERN ASSIGN INPUTS.PresSelCalStbd[9]:=(FALSE); editable
rectangle at (200,220)-(271,241): text "%.3f mA"; shows LS1905.Raw; alarm colour if LS1905.Err; runs INTERN ASSIGN INPUTS.PresSelCalStbd[9]:=(FALSE)
rectangle at (345,220)-(416,241): text "Off: %.3f"; shows LS1905.Cal_Off; runs INTERN ASSIGN INPUTS.PresSelCalStbd[9]:=(FALSE); editable
rectangle at (420,220)-(491,241): text "%.1f %%"; shows LS1905.Pos; runs INTERN ASSIGN INPUTS.PresSelCalStbd[9]:=(FALSE)
rectangle at (520,205)-(591,221): text "READ 0%"
rectangle at (595,205)-(666,221): text "READ 100%"
rounded rectangle at (685,250)-(756,271): text "APPLY"; toggles LS2005.Cal_Apply
rectangle at (595,250)-(666,271): text "%.3f V"; shows LS2005.Cal_Max; alarm colour if LS2005.Cal_Max = 0.0; runs INTERN ASSIGN INPUTS.PresSelCalStbd[9]:=(FALSE); editable
rectangle at (520,250)-(591,271): text "%.3f V"; shows LS2005.Cal_Min; alarm colour if LS2005.Cal_Min = 0.0; runs INTERN ASSIGN INPUTS.PresSelCalStbd[9]:=(FALSE); editable
rectangle at (45,250)-(191,271): text "Scoop AF PORT - LS2005"
rectangle at (275,250)-(346,271): text "K: %.3f"; shows LS2005.Cal_K; runs INTERN ASSIGN INPUTS.PresSelCalStbd[9]:=(FALSE); editable
rectangle at (200,250)-(271,271): text "%.3f V"; shows LS2005.Raw; alarm colour if LS2005.Err; runs INTERN ASSIGN INPUTS.PresSelCalStbd[9]:=(FALSE)
rectangle at (345,250)-(416,271): text "Off: %.3f"; shows LS2005.Cal_Off; runs INTERN ASSIGN INPUTS.PresSelCalStbd[9]:=(FALSE); editable
rectangle at (420,250)-(491,271): text "%.1f %%"; shows LS2005.Pos; runs INTERN ASSIGN INPUTS.PresSelCalStbd[9]:=(FALSE)
rounded rectangle at (685,280)-(756,301): text "APPLY"; toggles LS2201.Cal_Apply
rectangle at (595,280)-(666,301): text "%.3f mA"; shows LS2201.Cal_Max; alarm colour if LS2201.Cal_Max = 0.0; runs INTERN ASSIGN INPUTS.PresSelCalStbd[9]:=(FALSE); editable
rectangle at (520,280)-(591,301): text "%.3f mA"; shows LS2201.Cal_Min; alarm colour if LS2201.Cal_Min = 0.0; runs INTERN ASSIGN INPUTS.PresSelCalStbd[9]:=(FALSE); editable
rectangle at (45,280)-(191,301): text "Scoop UD STBD - LS2201"
rectangle at (275,280)-(346,301): text "K: %.3f"; shows LS2201.Cal_K; runs INTERN ASSIGN INPUTS.PresSelCalStbd[9]:=(FALSE); editable
rectangle at (200,280)-(271,301): text "%.3f mA"; shows LS2201.Raw; alarm colour if LS2201.Err; runs INTERN ASSIGN INPUTS.PresSelCalStbd[9]:=(FALSE)
rectangle at (345,280)-(416,301): text "Off: %.3f"; shows LS2201.Cal_Off; runs INTERN ASSIGN INPUTS.PresSelCalStbd[9]:=(FALSE); editable
rectangle at (420,280)-(491,301): text "%.1f %%"; shows LS2201.Pos; runs INTERN ASSIGN INPUTS.PresSelCalStbd[9]:=(FALSE)
rounded rectangle at (685,310)-(756,331): text "APPLY"; toggles LS2401.Cal_Apply
rectangle at (595,310)-(666,331): text "%.3f V"; shows LS2401.Cal_Max; alarm colour if LS2401.Cal_Max = 0.0; runs INTERN ASSIGN INPUTS.PresSelCalStbd[9]:=(FALSE); editable
rectangle at (520,310)-(591,331): text "%.3f V"; shows LS2401.Cal_Min; alarm colour if LS2401.Cal_Min = 0.0; runs INTERN ASSIGN INPUTS.PresSelCalStbd[9]:=(FALSE); editable
rectangle at (45,310)-(191,331): text "Scoop AF STBD - LS2401"
rectangle at (275,310)-(346,331): text "K: %.3f"; shows LS2401.Cal_K; runs INTERN ASSIGN INPUTS.PresSelCalStbd[9]:=(FALSE); editable
rectangle at (200,310)-(271,331): text "%.3f V"; shows LS2401.Raw; alarm colour if LS2401.Err; runs INTERN ASSIGN INPUTS.PresSelCalStbd[9]:=(FALSE)
rectangle at (345,310)-(416,331): text "Off: %.3f"; shows LS2401.Cal_Off; runs INTERN ASSIGN INPUTS.PresSelCalStbd[9]:=(FALSE); editable
rectangle at (420,310)-(491,331): text "%.1f %%"; shows LS2401.Pos; runs INTERN ASSIGN INPUTS.PresSelCalStbd[9]:=(FALSE)
rounded rectangle at (685,360)-(756,381): text "APPLY"; toggles LS2001.Cal_Apply
rectangle at (595,360)-(666,381): text "%.3f mA"; shows LS2001.Cal_Max; alarm colour if LS2001.Cal_Max = 0.0; runs INTERN ASSIGN INPUTS.PresSelCalStbd[9]:=(FALSE); editable
rectangle at (520,360)-(591,381): text "%.3f mA"; shows LS2001.Cal_Min; alarm colour if LS2001.Cal_Min = 0.0; runs INTERN ASSIGN INPUTS.PresSelCalStbd[9]:=(FALSE); editable
rectangle at (45,360)-(191,381): text "Valve C - LS2001"
rectangle at (275,360)-(346,381): text "K: %.3f"; shows LS2001.Cal_K; runs INTERN ASSIGN INPUTS.PresSelCalStbd[9]:=(FALSE); editable
rectangle at (200,360)-(271,381): text "%.3f mA"; shows LS2001.Raw; alarm colour if LS2001.Err; runs INTERN ASSIGN INPUTS.PresSelCalStbd[9]:=(FALSE)
rectangle at (345,360)-(416,381): text "Off: %.3f"; shows LS2001.Cal_Off; runs INTERN ASSIGN INPUTS.PresSelCalStbd[9]:=(FALSE); editable
rectangle at (420,360)-(491,381): text "%.1f %%"; shows LS2001.Pos; runs INTERN ASSIGN INPUTS.PresSelCalStbd[9]:=(FALSE)
rectangle at (520,345)-(591,361): text "READ 0%"
rectangle at (595,345)-(666,361): text "READ 100%"
rounded rectangle at (685,390)-(756,411): text "APPLY"; toggles LS2301.Cal_Apply
rectangle at (595,390)-(666,411): text "%.3f mA"; shows LS2301.Cal_Max; alarm colour if LS2301.Cal_Max = 0.0; runs INTERN ASSIGN INPUTS.PresSelCalStbd[9]:=(FALSE); editable
rectangle at (520,390)-(591,411): text "%.3f mA"; shows LS2301.Cal_Min; alarm colour if LS2301.Cal_Min = 0.0; runs INTERN ASSIGN INPUTS.PresSelCalStbd[9]:=(FALSE); editable
rectangle at (45,390)-(191,411): text "Valve S - LS2301"
rectangle at (275,390)-(346,411): text "K: %.3f"; shows LS2301.Cal_K; runs INTERN ASSIGN INPUTS.PresSelCalStbd[9]:=(FALSE); editable
rectangle at (200,390)-(271,411): text "%.3f mA"; shows LS2301.Raw; alarm colour if LS2301.Err; runs INTERN ASSIGN INPUTS.PresSelCalStbd[9]:=(FALSE)
rectangle at (345,390)-(416,411): text "Off: %.3f"; shows LS2301.Cal_Off; runs INTERN ASSIGN INPUTS.PresSelCalStbd[9]:=(FALSE); editable
rectangle at (420,390)-(491,411): text "%.1f %%"; shows LS2301.Pos; runs INTERN ASSIGN INPUTS.PresSelCalStbd[9]:=(FALSE)
rounded rectangle at (685,420)-(756,441): text "APPLY"; toggles LS2305.Cal_Apply
rectangle at (595,420)-(666,441): text "%.3f mA"; shows LS2305.Cal_Max; alarm colour if LS2305.Cal_Max = 0.0; runs INTERN ASSIGN INPUTS.PresSelCalStbd[9]:=(FALSE); editable
rectangle at (520,420)-(591,441): text "%.3f mA"; shows LS2305.Cal_Min; alarm colour if LS2305.Cal_Min = 0.0; runs INTERN ASSIGN INPUTS.PresSelCalStbd[9]:=(FALSE); editable
rectangle at (45,420)-(191,441): text "Valve B - LS2305"
rectangle at (275,420)-(346,441): text "K: %.3f"; shows LS2305.Cal_K; runs INTERN ASSIGN INPUTS.PresSelCalStbd[9]:=(FALSE); editable
rectangle at (200,420)-(271,441): text "%.3f mA"; shows LS2305.Raw; alarm colour if LS2305.Err; runs INTERN ASSIGN INPUTS.PresSelCalStbd[9]:=(FALSE)
rectangle at (345,420)-(416,441): text "Off: %.3f"; shows LS2305.Cal_Off; runs INTERN ASSIGN INPUTS.PresSelCalStbd[9]:=(FALSE); editable
rectangle at (420,420)-(491,441): text "%.1f %%"; shows LS2305.Pos; runs INTERN ASSIGN INPUTS.PresSelCalStbd[9]:=(FALSE)
rounded rectangle at (685,450)-(756,471): text "APPLY"; toggles LS2409.Cal_Apply
rectangle at (595,450)-(666,471): text "%.3f mA"; shows LS2409.Cal_Max; alarm colour if LS2409.Cal_Max = 0.0; runs INTERN ASSIGN INPUTS.PresSelCalStbd[9]:=(FALSE); editable
rectangle at (520,450)-(591,471): text "%.3f mA"; shows LS2409.Cal_Min; alarm colour if LS2409.Cal_Min = 0.0; runs INTERN ASSIGN INPUTS.PresSelCalStbd[9]:=(FALSE); editable
rectangle at (45,450)-(191,471): text "Valve R - LS2409"
rectangle at (275,450)-(346,471): text "K: %.3f"; shows LS2409.Cal_K; runs INTERN ASSIGN INPUTS.PresSelCalStbd[9]:=(FALSE); editable
rectangle at (200,450)-(271,471): text "%.3f mA"; shows LS2409.Raw; alarm colour if LS2409.Err; runs INTERN ASSIGN INPUTS.PresSelCalStbd[9]:=(FALSE)
rectangle at (345,450)-(416,471): text "Off: %.3f"; shows LS2409.Cal_Off; runs INTERN ASSIGN INPUTS.PresSelCalStbd[9]:=(FALSE); editable
rectangle at (420,450)-(491,471): text "%.1f %%"; shows LS2409.Pos; runs INTERN ASSIGN INPUTS.PresSelCalStbd[9]:=(FALSE)
rounded rectangle at (685,480)-(756,501): text "APPLY"; toggles LS2501.Cal_Apply
rectangle at (595,480)-(666,501): text "%.3f mA"; shows LS2501.Cal_Max; alarm colour if LS2501.Cal_Max = 0.0; runs INTERN ASSIGN INPUTS.PresSelCalStbd[9]:=(FALSE); editable
rectangle at (520,480)-(591,501): text "%.3f mA"; shows LS2501.Cal_Min; alarm colour if LS2501.Cal_Min = 0.0; runs INTERN ASSIGN INPUTS.PresSelCalStbd[9]:=(FALSE); editable
rectangle at (45,480)-(191,501): text "Valve N - LS2501"
rectangle at (275,480)-(346,501): text "K: %.3f"; shows LS2501.Cal_K; runs INTERN ASSIGN INPUTS.PresSelCalStbd[9]:=(FALSE); editable
rectangle at (200,480)-(271,501): text "%.3f mA"; shows LS2501.Raw; alarm colour if LS2501.Err; runs INTERN ASSIGN INPUTS.PresSelCalStbd[9]:=(FALSE)
rectangle at (345,480)-(416,501): text "Off: %.3f"; shows LS2501.Cal_Off; runs INTERN ASSIGN INPUTS.PresSelCalStbd[9]:=(FALSE); editable
rectangle at (420,480)-(491,501): text "%.1f %%"; shows LS2501.Pos; runs INTERN ASSIGN INPUTS.PresSelCalStbd[9]:=(FALSE)
rounded rectangle at (685,510)-(756,531): text "APPLY"; toggles LS2505.Cal_Apply
rectangle at (595,510)-(666,531): text "%.3f mA"; shows LS2505.Cal_Max; alarm colour if LS2505.Cal_Max = 0.0; runs INTERN ASSIGN INPUTS.PresSelCalStbd[9]:=(FALSE); editable
rectangle at (520,510)-(591,531): text "%.3f mA"; shows LS2505.Cal_Min; alarm colour if LS2505.Cal_Min = 0.0; runs INTERN ASSIGN INPUTS.PresSelCalStbd[9]:=(FALSE); editable
rectangle at (45,510)-(191,531): text "Valve I - LS2505"
rectangle at (275,510)-(346,531): text "K: %.3f"; shows LS2505.Cal_K; runs INTERN ASSIGN INPUTS.PresSelCalStbd[9]:=(FALSE); editable
rectangle at (200,510)-(271,531): text "%.3f mA"; shows LS2505.Raw; alarm colour if LS2505.Err; runs INTERN ASSIGN INPUTS.PresSelCalStbd[9]:=(FALSE)
rectangle at (345,510)-(416,531): text "Off: %.3f"; shows LS2505.Cal_Off; runs INTERN ASSIGN INPUTS.PresSelCalStbd[9]:=(FALSE); editable
rectangle at (420,510)-(491,531): text "%.1f %%"; shows LS2505.Pos; runs INTERN ASSIGN INPUTS.PresSelCalStbd[9]:=(FALSE)
rectangle at (770,360)-(881,381): text "(OPEN  -> 100%)"
rectangle at (770,390)-(881,411): text "(OPEN  -> 100%)"
rectangle at (770,420)-(881,441): text "(OPEN  -> 100%)"
rectangle at (770,450)-(881,471): text "(OPEN  -> 100%)"
rectangle at (770,480)-(881,501): text "(OPEN  -> 100%)"
rectangle at (770,510)-(881,531): text "(OPEN  -> 100%)"
rectangle at (770,220)-(891,241): text "(DW/OPEN -> 100%)"
rectangle at (770,280)-(891,301): text "(DW/OPEN  -> 100%)"
rectangle at (770,250)-(891,271): text "(AFT -> 100%)"
rectangle at (770,310)-(891,331): text "(AFT -> 100%)"
19 more shapes without text or variables
*)

(* Visualisation VISU_CFG_BOARD
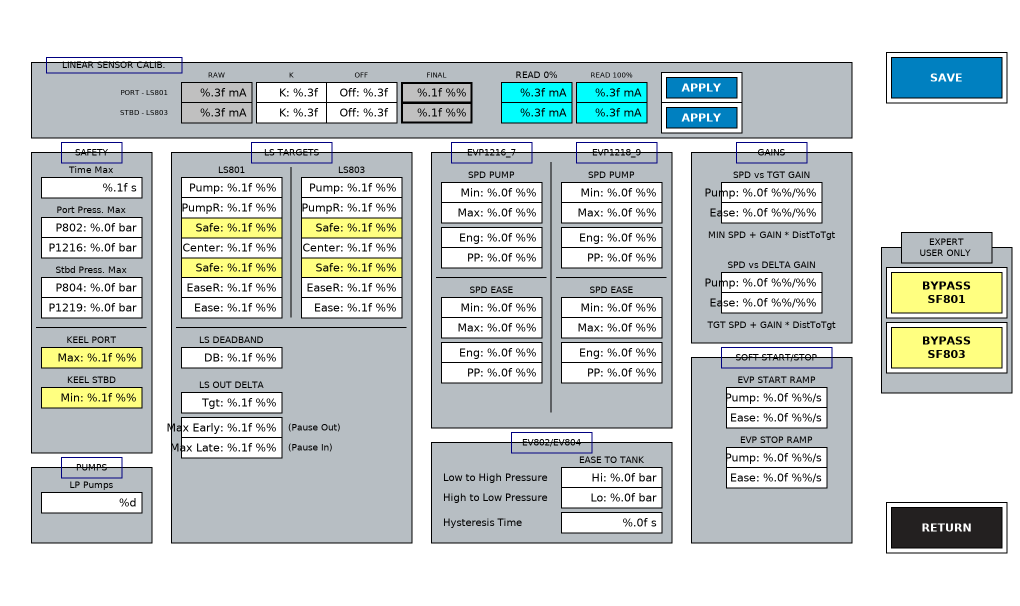
rectangle at (265,140)-(346,161): text "LS TARGETS"
rectangle at (75,140)-(136,161): text "SAFETY"
rectangle at (60,55)-(196,71): text "LINEAR SENSOR CALIB."
rectangle at (415,65)-(486,81): text "FINAL"
rectangle at (20,550)-(331,601): text "%s"; shows INPUTS.sVisuTime
rounded rectangle at (905,55)-(1016,96): text "SAVE"; alarm colour if PARAMS.Save; toggles PARAMS.Save
rounded rectangle at (905,505)-(1016,546): text "RETURN"; opens VISU_2_BOARD
rectangle at (730,550)-(896,601): text "SAVED!"; invisible if PARAMS.Saved
rectangle at (20,0)-(426,51): text "CFG: BOARD"
rounded rectangle at (680,75)-(751,96): text "APPLY"; toggles LS801.Cal_Apply
rectangle at (590,80)-(661,101): text "%.3f mA"; shows LS801.Cal_Max; alarm colour if LS801.Cal_Max = 0.0; runs INTERN ASSIGN INPUTS.PresSelCalStbd[9]:=(FALSE); editable
rectangle at (515,80)-(586,101): text "%.3f mA"; shows LS801.Cal_Min; alarm colour if LS801.Cal_Min = 0.0; runs INTERN ASSIGN INPUTS.PresSelCalStbd[9]:=(FALSE); editable
rectangle at (50,80)-(186,101): text "PORT - LS801"
rectangle at (270,80)-(341,101): text "K: %.3f"; shows LS801.Cal_K; runs INTERN ASSIGN INPUTS.PresSelCalStbd[9]:=(FALSE); editable
rectangle at (195,80)-(266,101): text "%.3f mA"; shows LS801.Raw; alarm colour if LS801.Err; runs INTERN ASSIGN INPUTS.PresSelCalStbd[9]:=(FALSE)
rectangle at (340,80)-(411,101): text "Off: %.3f"; shows LS801.Cal_Off; runs INTERN ASSIGN INPUTS.PresSelCalStbd[9]:=(FALSE); editable
rectangle at (415,80)-(486,101): text "%.1f %%"; shows LS801.Pos; runs INTERN ASSIGN INPUTS.PresSelCalStbd[9]:=(FALSE)
rectangle at (515,65)-(586,81): text "READ 0%"
rectangle at (590,65)-(661,81): text "READ 100%"
rounded rectangle at (680,105)-(751,126): text "APPLY"; toggles LS803.Cal_Apply
rectangle at (590,100)-(661,121): text "%.3f mA"; shows LS803.Cal_Max; alarm colour if LS803.Cal_Max = 0.0; runs INTERN ASSIGN INPUTS.PresSelCalStbd[9]:=(FALSE); editable
rectangle at (515,100)-(586,121): text "%.3f mA"; shows LS803.Cal_Min; alarm colour if LS803.Cal_Min = 0.0; runs INTERN ASSIGN INPUTS.PresSelCalStbd[9]:=(FALSE); editable
rectangle at (50,100)-(186,121): text "STBD - LS803"
rectangle at (270,100)-(341,121): text "K: %.3f"; shows LS803.Cal_K; runs INTERN ASSIGN INPUTS.PresSelCalStbd[9]:=(FALSE); editable
rectangle at (195,100)-(266,121): text "%.3f mA"; shows LS803.Raw; alarm colour if LS803.Err; runs INTERN ASSIGN INPUTS.PresSelCalStbd[9]:=(FALSE)
rectangle at (340,100)-(411,121): text "Off: %.3f"; shows LS803.Cal_Off; runs INTERN ASSIGN INPUTS.PresSelCalStbd[9]:=(FALSE); editable
rectangle at (415,100)-(486,121): text "%.1f %%"; shows LS803.Pos; runs INTERN ASSIGN INPUTS.PresSelCalStbd[9]:=(FALSE)
rectangle at (55,215)-(156,236): text "P802: %.0f bar"; shows P802.MaxBar; runs INTERN ASSIGN INPUTS.PresSelCalStbd[9]:=(FALSE); editable
rectangle at (55,200)-(156,216): text "Port Press. Max"
rectangle at (55,275)-(156,296): text "P804: %.0f bar"; shows P804.MaxBar; runs INTERN ASSIGN INPUTS.PresSelCalStbd[9]:=(FALSE); editable
rectangle at (55,175)-(156,196): text "%.1f s"; shows PARAMS.stBoardCfg.TimeMax; runs INTERN ASSIGN INPUTS.PresSelCalStbd[9]:=(FALSE); editable
rectangle at (65,160)-(146,176): text "Time Max"
rectangle at (55,490)-(156,511): text "%d"; shows PARAMS.stBoardCfg.LP; runs INTERN ASSIGN INPUTS.PresSelCalStbd[9]:=(FALSE); editable 1..2
rectangle at (55,475)-(156,491): text "LP Pumps"
rectangle at (455,180)-(556,201): text "Min: %.0f %%"; shows PARAMS.stBoardCfg.EVP_In_P_Min; runs INTERN ASSIGN INPUTS.PresSelCalStbd[9]:=(FALSE); editable
rectangle at (455,165)-(556,181): text "SPD PUMP"
rectangle at (455,200)-(556,221): text "Max: %.0f %%"; shows PARAMS.stBoardCfg.EVP_In_P_Max; runs INTERN ASSIGN INPUTS.PresSelCalStbd[9]:=(FALSE); editable
rectangle at (455,295)-(556,316): text "Min: %.0f %%"; shows PARAMS.stBoardCfg.EVP_Out_P_Min; runs INTERN ASSIGN INPUTS.PresSelCalStbd[9]:=(FALSE); editable
rectangle at (455,280)-(556,296): text "SPD EASE"
rectangle at (455,315)-(556,336): text "Max: %.0f %%"; shows PARAMS.stBoardCfg.EVP_Out_P_Max; runs INTERN ASSIGN INPUTS.PresSelCalStbd[9]:=(FALSE); editable
rectangle at (575,180)-(676,201): text "Min: %.0f %%"; shows PARAMS.stBoardCfg.EVP_In_S_Min; runs INTERN ASSIGN INPUTS.PresSelCalStbd[9]:=(FALSE); editable
rectangle at (575,165)-(676,181): text "SPD PUMP"
rectangle at (575,200)-(676,221): text "Max: %.0f %%"; shows PARAMS.stBoardCfg.EVP_In_S_Max; runs INTERN ASSIGN INPUTS.PresSelCalStbd[9]:=(FALSE); editable
rectangle at (575,295)-(676,316): text "Min: %.0f %%"; shows PARAMS.stBoardCfg.EVP_Out_S_Min; runs INTERN ASSIGN INPUTS.PresSelCalStbd[9]:=(FALSE); editable
rectangle at (575,280)-(676,296): text "SPD EASE"
rectangle at (575,315)-(676,336): text "Max: %.0f %%"; shows PARAMS.stBoardCfg.EVP_Out_S_Max; runs INTERN ASSIGN INPUTS.PresSelCalStbd[9]:=(FALSE); editable
rectangle at (55,260)-(156,276): text "Stbd Press. Max"
rectangle at (55,235)-(156,256): text "P1216: %.0f bar"; shows P1216.MaxBar; runs INTERN ASSIGN INPUTS.PresSelCalStbd[9]:=(FALSE); editable
rectangle at (55,295)-(156,316): text "P1219: %.0f bar"; shows P1219.MaxBar; runs INTERN ASSIGN INPUTS.PresSelCalStbd[9]:=(FALSE); editable
rectangle at (455,225)-(556,246): text "Eng: %.0f %%"; shows PARAMS.stBoardCfg.EVP_In_P_Eng; runs INTERN ASSIGN INPUTS.PresSelCalStbd[9]:=(FALSE); editable
rectangle at (455,245)-(556,266): text "PP: %.0f %%"; shows PARAMS.stBoardCfg.EVP_In_P_PP; runs INTERN ASSIGN INPUTS.PresSelCalStbd[9]:=(FALSE); editable
rectangle at (575,225)-(676,246): text "Eng: %.0f %%"; shows PARAMS.stBoardCfg.EVP_In_S_Eng; runs INTERN ASSIGN INPUTS.PresSelCalStbd[9]:=(FALSE); editable
rectangle at (575,245)-(676,266): text "PP: %.0f %%"; shows PARAMS.stBoardCfg.EVP_In_S_PP; runs INTERN ASSIGN INPUTS.PresSelCalStbd[9]:=(FALSE); editable
rectangle at (455,340)-(556,361): text "Eng: %.0f %%"; shows PARAMS.stBoardCfg.EVP_Out_P_Eng; runs INTERN ASSIGN INPUTS.PresSelCalStbd[9]:=(FALSE); editable
rectangle at (455,360)-(556,381): text "PP: %.0f %%"; shows PARAMS.stBoardCfg.EVP_Out_P_PP; runs INTERN ASSIGN INPUTS.PresSelCalStbd[9]:=(FALSE); editable
rectangle at (575,340)-(676,361): text "Eng: %.0f %%"; shows PARAMS.stBoardCfg.EVP_Out_S_Eng; runs INTERN ASSIGN INPUTS.PresSelCalStbd[9]:=(FALSE); editable
rectangle at (575,360)-(676,381): text "PP: %.0f %%"; shows PARAMS.stBoardCfg.EVP_Out_S_PP; runs INTERN ASSIGN INPUTS.PresSelCalStbd[9]:=(FALSE); editable
rectangle at (740,385)-(841,406): text "Pump: %.0f %%/s"; shows PARAMS.stBoardCfg.EVP_In_Inc; runs INTERN ASSIGN INPUTS.PresSelCalStbd[9]:=(FALSE); editable
rectangle at (740,370)-(841,386): text "EVP START RAMP"
rectangle at (740,405)-(841,426): text "Ease: %.0f %%/s"; shows PARAMS.stBoardCfg.EVP_Out_Inc; runs INTERN ASSIGN INPUTS.PresSelCalStbd[9]:=(FALSE); editable
rectangle at (195,175)-(296,196): text "Pump: %.1f %%"; shows PARAMS.stBoardCfg.TgtLS_P_In; runs INTERN ASSIGN INPUTS.PresSelCalStbd[9]:=(FALSE); editable
rectangle at (195,160)-(296,176): text "LS801"
rectangle at (195,255)-(296,276): text "Safe: %.1f %%"; shows PARAMS.stBoardCfg.TgtLS_P_Safe_Out; runs INTERN ASSIGN INPUTS.PresSelCalStbd[9]:=(FALSE); editable
rectangle at (195,235)-(296,256): text "Center: %.1f %%"; shows PARAMS.stBoardCfg.TgtLS_P_Mid; runs INTERN ASSIGN INPUTS.PresSelCalStbd[9]:=(FALSE); editable
rectangle at (195,215)-(296,236): text "Safe: %.1f %%"; shows PARAMS.stBoardCfg.TgtLS_P_Safe_In; runs INTERN ASSIGN INPUTS.PresSelCalStbd[9]:=(FALSE); editable
rectangle at (195,275)-(296,296): text "EaseR: %.1f %%"; shows PARAMS.stBoardCfg.TgtLS_P_OutR; runs INTERN ASSIGN INPUTS.PresSelCalStbd[9]:=(FALSE); editable
rectangle at (195,345)-(296,366): text "DB: %.1f %%"; shows PARAMS.stBoardCfg.LS_DB; runs INTERN ASSIGN INPUTS.PresSelCalStbd[9]:=(FALSE); editable
rectangle at (195,330)-(296,346): text "LS DEADBAND"
rectangle at (195,390)-(296,411): text "Tgt: %.1f %%"; shows PARAMS.stBoardCfg.LS_Dif_Tgt; runs INTERN ASSIGN INPUTS.PresSelCalStbd[9]:=(FALSE); editable
rectangle at (195,375)-(296,391): text "LS OUT DELTA"
rectangle at (735,180)-(836,201): text "Pump: %.0f %%/%%"; shows PARAMS.stBoardCfg.EVP_In_LS_K; runs INTERN ASSIGN INPUTS.PresSelCalStbd[9]:=(FALSE); editable
rectangle at (735,165)-(836,181): text "SPD vs TGT GAIN"
rectangle at (735,200)-(836,221): text "Ease: %.0f %%/%%"; shows PARAMS.stBoardCfg.EVP_Out_LS_K; runs INTERN ASSIGN INPUTS.PresSelCalStbd[9]:=(FALSE); editable
rectangle at (735,270)-(836,291): text "Pump: %.0f %%/%%"; shows PARAMS.stBoardCfg.EVP_In_EVP_K; runs INTERN ASSIGN INPUTS.PresSelCalStbd[9]:=(FALSE); editable
rectangle at (730,255)-(841,271): text "SPD vs DELTA GAIN"
rectangle at (735,290)-(836,311): text "Ease: %.0f %%/%%"; shows PARAMS.stBoardCfg.EVP_Out_EVP_K; runs INTERN ASSIGN INPUTS.PresSelCalStbd[9]:=(FALSE); editable
rectangle at (315,175)-(416,196): text "Pump: %.1f %%"; shows PARAMS.stBoardCfg.TgtLS_S_In; runs INTERN ASSIGN INPUTS.PresSelCalStbd[9]:=(FALSE); editable
rectangle at (315,160)-(416,176): text "LS803"
rectangle at (315,255)-(416,276): text "Safe: %.1f %%"; shows PARAMS.stBoardCfg.TgtLS_S_Safe_Out; runs INTERN ASSIGN INPUTS.PresSelCalStbd[9]:=(FALSE); editable
rectangle at (315,235)-(416,256): text "Center: %.1f %%"; shows PARAMS.stBoardCfg.TgtLS_S_Mid; runs INTERN ASSIGN INPUTS.PresSelCalStbd[9]:=(FALSE); editable
rectangle at (315,215)-(416,236): text "Safe: %.1f %%"; shows PARAMS.stBoardCfg.TgtLS_S_Safe_In; runs INTERN ASSIGN INPUTS.PresSelCalStbd[9]:=(FALSE); editable
rectangle at (315,275)-(416,296): text "EaseR: %.1f %%"; shows PARAMS.stBoardCfg.TgtLS_S_OutR; runs INTERN ASSIGN INPUTS.PresSelCalStbd[9]:=(FALSE); editable
rectangle at (55,345)-(156,366): text "Max: %.1f %%"; shows PARAMS.stBoardCfg.Keel_P_Max; runs INTERN ASSIGN INPUTS.PresSelCalStbd[9]:=(FALSE); editable
rectangle at (55,330)-(156,346): text "KEEL PORT"
rectangle at (55,385)-(156,406): text "Min: %.1f %%"; shows PARAMS.stBoardCfg.Keel_S_Min; runs INTERN ASSIGN INPUTS.PresSelCalStbd[9]:=(FALSE); editable
rectangle at (55,370)-(156,386): text "KEEL STBD"
rectangle at (195,415)-(296,436): text "Max Early: %.1f %%"; shows PARAMS.stBoardCfg.LS_Dif_Max; runs INTERN ASSIGN INPUTS.PresSelCalStbd[9]:=(FALSE); editable
rectangle at (195,435)-(296,456): text "Max Late: %.1f %%"; shows PARAMS.stBoardCfg.LS_Dif_Min; runs INTERN ASSIGN INPUTS.PresSelCalStbd[9]:=(FALSE); editable
rectangle at (300,415)-(371,436): text "(Pause Out)"
rectangle at (300,435)-(371,456): text "(Pause In)"
rectangle at (710,225)-(861,241): text "MIN SPD + GAIN * DistToTgt"
rectangle at (740,445)-(841,466): text "Pump: %.0f %%/s"; shows PARAMS.stBoardCfg.EVP_In_Dec; runs INTERN ASSIGN INPUTS.PresSelCalStbd[9]:=(FALSE); editable
rectangle at (740,430)-(841,446): text "EVP STOP RAMP"
rectangle at (740,465)-(841,486): text "Ease: %.0f %%/s"; shows PARAMS.stBoardCfg.EVP_Out_Dec; runs INTERN ASSIGN INPUTS.PresSelCalStbd[9]:=(FALSE); editable
rectangle at (575,465)-(676,486): text "Hi: %.0f bar"; shows PARAMS.stBoardCfg.P_Hyst_HP; runs INTERN ASSIGN INPUTS.PresSelCalStbd[9]:=(FALSE); editable
rectangle at (575,485)-(676,506): text "Lo: %.0f bar"; shows PARAMS.stBoardCfg.P_Hyst_LP; runs INTERN ASSIGN INPUTS.PresSelCalStbd[9]:=(FALSE); editable
rectangle at (575,510)-(676,531): text "%.0f s"; shows PARAMS.stBoardCfg.P_Hyst_TM; runs INTERN ASSIGN INPUTS.PresSelCalStbd[9]:=(FALSE); editable
rectangle at (455,465)-(571,486): text "Low to High Pressure"; shows RECV_J1939.F004.DriverDemandTorque
rectangle at (455,485)-(571,506): text "High to Low Pressure"; shows RECV_J1939.F004.DriverDemandTorque
rectangle at (455,510)-(571,531): text "Hysteresis Time"; shows RECV_J1939.F004.DriverDemandTorque
rectangle at (575,450)-(676,466): text "EASE TO TANK"
rectangle at (195,65)-(266,81): text "RAW"
rectangle at (270,65)-(341,81): text "K"
rectangle at (340,65)-(411,81): text "OFF"
rectangle at (465,140)-(546,161): text "EVP1216_7"
rectangle at (710,315)-(861,331): text "TGT SPD + GAIN * DistToTgt"
rectangle at (590,140)-(671,161): text "EVP1218_9"
rectangle at (750,140)-(821,161): text "GAINS"
rounded rectangle at (525,430)-(606,451): text "EV802/EV804"
rectangle at (75,455)-(136,476): text "PUMPS"
rectangle at (735,345)-(846,366): text "SOFT START/STOP"
rectangle at (195,195)-(296,216): text "PumpR: %.1f %%"; shows PARAMS.stBoardCfg.TgtLS_P_InR; runs INTERN ASSIGN INPUTS.PresSelCalStbd[9]:=(FALSE); editable
rectangle at (315,195)-(416,216): text "PumpR: %.1f %%"; shows PARAMS.stBoardCfg.TgtLS_S_InR; runs INTERN ASSIGN INPUTS.PresSelCalStbd[9]:=(FALSE); editable
rectangle at (195,295)-(296,316): text "Ease: %.1f %%"; shows PARAMS.stBoardCfg.TgtLS_P_Out; runs INTERN ASSIGN INPUTS.PresSelCalStbd[9]:=(FALSE); editable
rectangle at (315,295)-(416,316): text "Ease: %.1f %%"; shows PARAMS.stBoardCfg.TgtLS_S_Out; runs INTERN ASSIGN INPUTS.PresSelCalStbd[9]:=(FALSE); editable
rounded rectangle at (915,230)-(1006,261): text "EXPERT / USER ONLY"
rounded rectangle at (905,270)-(1016,311): text "BYPASS / SF801"
rounded rectangle at (905,325)-(1016,366): text "BYPASS / SF803"
21 more shapes without text or variables
*)

(* Visualisation VISU_CFG_CYLINDERS1
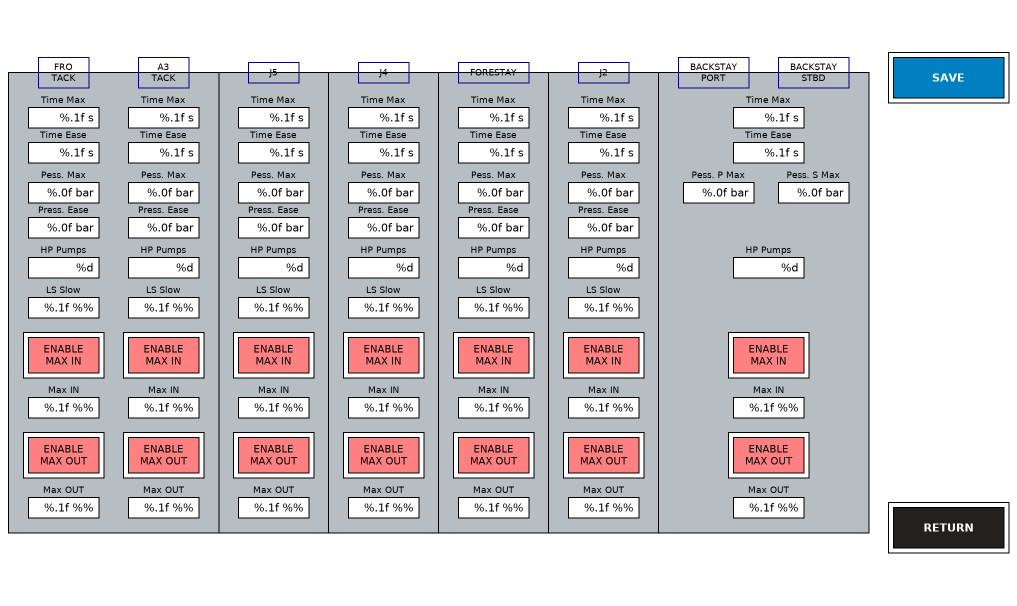
rectangle at (20,550)-(331,601): text "%s"; shows INPUTS.sVisuTime
rounded rectangle at (905,505)-(1016,546): text "RETURN"; opens VISU_1_CYLINDERS1
rectangle at (730,550)-(896,601): text "SAVED!"; invisible if PARAMS.Saved
rectangle at (40,395)-(111,416): text "%.1f %%"; shows PARAMS.stSE301Cfg.TgtLS_In; runs INTERN ASSIGN INPUTS.PresSelCalStbd[9]:=(FALSE); editable
rectangle at (40,90)-(111,106): text "Time Max"
rectangle at (40,380)-(111,396): text "Max IN"
rectangle at (40,165)-(111,181): text "Pess. Max"
rectangle at (40,215)-(111,236): text "%.0f bar"; shows PARAMS.stSE301Cfg.Ease; runs INTERN ASSIGN INPUTS.PresSelCalStbd[9]:=(FALSE); editable
rectangle at (40,200)-(111,216): text "Press. Ease"
rectangle at (40,495)-(111,516): text "%.1f %%"; shows PARAMS.stSE301Cfg.TgtLS_Out; runs INTERN ASSIGN INPUTS.PresSelCalStbd[9]:=(FALSE); editable
rectangle at (40,480)-(111,496): text "Max OUT"
rectangle at (40,140)-(111,161): text "%.1f s"; shows PARAMS.stSE301Cfg.TimeEase; runs INTERN ASSIGN INPUTS.PresSelCalStbd[9]:=(FALSE); editable
rectangle at (40,125)-(111,141): text "Time Ease"
rectangle at (40,255)-(111,276): text "%d"; shows PARAMS.stSE301Cfg.HP; runs INTERN ASSIGN INPUTS.PresSelCalStbd[9]:=(FALSE); editable 1..2
rectangle at (40,240)-(111,256): text "HP Pumps"
rounded rectangle at (40,335)-(111,371): text "ENABLE / MAX IN"; alarm colour if PARAMS.stSE301Cfg.LS_Limit_In; toggles PARAMS.stSE301Cfg.LS_Limit_In
rounded rectangle at (40,435)-(111,471): text "ENABLE / MAX OUT"; alarm colour if PARAMS.stSE301Cfg.LS_Limit_Out; toggles PARAMS.stSE301Cfg.LS_Limit_Out
rectangle at (140,395)-(211,416): text "%.1f %%"; shows PARAMS.stSE303Cfg.TgtLS_In; runs INTERN ASSIGN INPUTS.PresSelCalStbd[9]:=(FALSE); editable
rectangle at (140,215)-(211,236): text "%.0f bar"; shows PARAMS.stSE303Cfg.Ease; runs INTERN ASSIGN INPUTS.PresSelCalStbd[9]:=(FALSE); editable
rectangle at (140,495)-(211,516): text "%.1f %%"; shows PARAMS.stSE303Cfg.TgtLS_Out; runs INTERN ASSIGN INPUTS.PresSelCalStbd[9]:=(FALSE); editable
rectangle at (140,140)-(211,161): text "%.1f s"; shows PARAMS.stSE303Cfg.TimeEase; runs INTERN ASSIGN INPUTS.PresSelCalStbd[9]:=(FALSE); editable
rectangle at (140,255)-(211,276): text "%d"; shows PARAMS.stSE303Cfg.HP; runs INTERN ASSIGN INPUTS.PresSelCalStbd[9]:=(FALSE); editable 1..2
rounded rectangle at (140,335)-(211,371): text "ENABLE / MAX IN"; alarm colour if PARAMS.stSE303Cfg.LS_Limit_In; toggles PARAMS.stSE303Cfg.LS_Limit_In
rounded rectangle at (140,435)-(211,471): text "ENABLE / MAX OUT"; alarm colour if PARAMS.stSE303Cfg.LS_Limit_Out; toggles PARAMS.stSE303Cfg.LS_Limit_Out
rectangle at (745,395)-(816,416): text "%.1f %%"; shows PARAMS.stSE901Cfg.TgtLS_In; runs INTERN ASSIGN INPUTS.PresSelCalStbd[9]:=(FALSE); editable
rectangle at (745,495)-(816,516): text "%.1f %%"; shows PARAMS.stSE901Cfg.TgtLS_Out; runs INTERN ASSIGN INPUTS.PresSelCalStbd[9]:=(FALSE); editable
rectangle at (745,140)-(816,161): text "%.1f s"; shows PARAMS.stSE901Cfg.TimeEase; runs INTERN ASSIGN INPUTS.PresSelCalStbd[9]:=(FALSE); editable
rectangle at (745,255)-(816,276): text "%d"; shows PARAMS.stSE901Cfg.HP; runs INTERN ASSIGN INPUTS.PresSelCalStbd[9]:=(FALSE); editable 1..2
rounded rectangle at (745,335)-(816,371): text "ENABLE / MAX IN"; alarm colour if PARAMS.stSE901Cfg.LS_Limit_In; toggles PARAMS.stSE901Cfg.LS_Limit_In
rounded rectangle at (745,435)-(816,471): text "ENABLE / MAX OUT"; alarm colour if PARAMS.stSE901Cfg.LS_Limit_Out; toggles PARAMS.stSE901Cfg.LS_Limit_Out
rectangle at (790,165)-(861,181): text "Pess. S Max"
rectangle at (20,0)-(426,51): text "CFG: CYLINDERS 1"
rectangle at (250,395)-(321,416): text "%.1f %%"; shows PARAMS.stSE305Cfg.TgtLS_In; runs INTERN ASSIGN INPUTS.PresSelCalStbd[9]:=(FALSE); editable
rectangle at (250,215)-(321,236): text "%.0f bar"; shows PARAMS.stSE305Cfg.Ease; runs INTERN ASSIGN INPUTS.PresSelCalStbd[9]:=(FALSE); editable
rectangle at (250,495)-(321,516): text "%.1f %%"; shows PARAMS.stSE305Cfg.TgtLS_Out; runs INTERN ASSIGN INPUTS.PresSelCalStbd[9]:=(FALSE); editable
rectangle at (250,140)-(321,161): text "%.1f s"; shows PARAMS.stSE305Cfg.TimeEase; runs INTERN ASSIGN INPUTS.PresSelCalStbd[9]:=(FALSE); editable
rectangle at (250,255)-(321,276): text "%d"; shows PARAMS.stSE305Cfg.HP; runs INTERN ASSIGN INPUTS.PresSelCalStbd[9]:=(FALSE); editable 1..2
rounded rectangle at (250,335)-(321,371): text "ENABLE / MAX IN"; alarm colour if PARAMS.stSE305Cfg.LS_Limit_In; toggles PARAMS.stSE305Cfg.LS_Limit_In
rounded rectangle at (250,435)-(321,471): text "ENABLE / MAX OUT"; alarm colour if PARAMS.stSE305Cfg.LS_Limit_Out; toggles PARAMS.stSE305Cfg.LS_Limit_Out
rectangle at (360,395)-(431,416): text "%.1f %%"; shows PARAMS.stSE307Cfg.TgtLS_In; runs INTERN ASSIGN INPUTS.PresSelCalStbd[9]:=(FALSE); editable
rectangle at (360,215)-(431,236): text "%.0f bar"; shows PARAMS.stSE307Cfg.Ease; runs INTERN ASSIGN INPUTS.PresSelCalStbd[9]:=(FALSE); editable
rectangle at (360,495)-(431,516): text "%.1f %%"; shows PARAMS.stSE307Cfg.TgtLS_Out; runs INTERN ASSIGN INPUTS.PresSelCalStbd[9]:=(FALSE); editable
rectangle at (360,140)-(431,161): text "%.1f s"; shows PARAMS.stSE307Cfg.TimeEase; runs INTERN ASSIGN INPUTS.PresSelCalStbd[9]:=(FALSE); editable
rectangle at (360,255)-(431,276): text "%d"; shows PARAMS.stSE307Cfg.HP; runs INTERN ASSIGN INPUTS.PresSelCalStbd[9]:=(FALSE); editable 1..2
rounded rectangle at (360,335)-(431,371): text "ENABLE / MAX IN"; alarm colour if PARAMS.stSE307Cfg.LS_Limit_In; toggles PARAMS.stSE307Cfg.LS_Limit_In
rounded rectangle at (360,435)-(431,471): text "ENABLE / MAX OUT"; alarm colour if PARAMS.stSE307Cfg.LS_Limit_Out; toggles PARAMS.stSE307Cfg.LS_Limit_Out
rectangle at (470,215)-(541,236): text "%.0f bar"; shows PARAMS.stSE309Cfg.Ease; runs INTERN ASSIGN INPUTS.PresSelCalStbd[9]:=(FALSE); editable
rectangle at (470,140)-(541,161): text "%.1f s"; shows PARAMS.stSE309Cfg.TimeEase; runs INTERN ASSIGN INPUTS.PresSelCalStbd[9]:=(FALSE); editable
rectangle at (470,255)-(541,276): text "%d"; shows PARAMS.stSE309Cfg.HP; runs INTERN ASSIGN INPUTS.PresSelCalStbd[9]:=(FALSE); editable 1..2
rectangle at (580,395)-(651,416): text "%.1f %%"; shows PARAMS.stSE311Cfg.TgtLS_In; runs INTERN ASSIGN INPUTS.PresSelCalStbd[9]:=(FALSE); editable
rectangle at (580,215)-(651,236): text "%.0f bar"; shows PARAMS.stSE311Cfg.Ease; runs INTERN ASSIGN INPUTS.PresSelCalStbd[9]:=(FALSE); editable
rectangle at (580,495)-(651,516): text "%.1f %%"; shows PARAMS.stSE311Cfg.TgtLS_Out; runs INTERN ASSIGN INPUTS.PresSelCalStbd[9]:=(FALSE); editable
rectangle at (580,140)-(651,161): text "%.1f s"; shows PARAMS.stSE311Cfg.TimeEase; runs INTERN ASSIGN INPUTS.PresSelCalStbd[9]:=(FALSE); editable
rectangle at (580,255)-(651,276): text "%d"; shows PARAMS.stSE311Cfg.HP; runs INTERN ASSIGN INPUTS.PresSelCalStbd[9]:=(FALSE); editable 1..2
rounded rectangle at (580,335)-(651,371): text "ENABLE / MAX IN"; alarm colour if PARAMS.stSE311Cfg.LS_Limit_In; toggles PARAMS.stSE311Cfg.LS_Limit_In
rounded rectangle at (580,435)-(651,471): text "ENABLE / MAX OUT"; alarm colour if PARAMS.stSE311Cfg.LS_Limit_Out; toggles PARAMS.stSE311Cfg.LS_Limit_Out
rectangle at (790,180)-(861,201): text "%.0f bar"; shows P903.MaxBar; runs INTERN ASSIGN INPUTS.PresSelCalStbd[9]:=(FALSE); editable
rectangle at (695,180)-(766,201): text "%.0f bar"; shows P901.MaxBar; runs INTERN ASSIGN INPUTS.PresSelCalStbd[9]:=(FALSE); editable
rectangle at (40,105)-(111,126): text "%.1f s"; shows PARAMS.stSE301Cfg.TimeMax; runs INTERN ASSIGN INPUTS.PresSelCalStbd[9]:=(FALSE); editable
rectangle at (140,105)-(211,126): text "%.1f s"; shows PARAMS.stSE303Cfg.TimeMax; runs INTERN ASSIGN INPUTS.PresSelCalStbd[9]:=(FALSE); editable
rectangle at (745,105)-(816,126): text "%.1f s"; shows PARAMS.stSE901Cfg.TimeMax; runs INTERN ASSIGN INPUTS.PresSelCalStbd[9]:=(FALSE); editable
rectangle at (250,105)-(321,126): text "%.1f s"; shows PARAMS.stSE305Cfg.TimeMax; runs INTERN ASSIGN INPUTS.PresSelCalStbd[9]:=(FALSE); editable
rectangle at (360,105)-(431,126): text "%.1f s"; shows PARAMS.stSE307Cfg.TimeMax; runs INTERN ASSIGN INPUTS.PresSelCalStbd[9]:=(FALSE); editable
rectangle at (470,105)-(541,126): text "%.1f s"; shows PARAMS.stSE309Cfg.TimeMax; runs INTERN ASSIGN INPUTS.PresSelCalStbd[9]:=(FALSE); editable
rectangle at (580,105)-(651,126): text "%.1f s"; shows PARAMS.stSE311Cfg.TimeMax; runs INTERN ASSIGN INPUTS.PresSelCalStbd[9]:=(FALSE); editable
rectangle at (40,180)-(111,201): text "%.0f bar"; shows P301.MaxBar; runs INTERN ASSIGN INPUTS.PresSelCalStbd[9]:=(FALSE); editable
rectangle at (140,180)-(211,201): text "%.0f bar"; shows P303.MaxBar; runs INTERN ASSIGN INPUTS.PresSelCalStbd[9]:=(FALSE); editable
rectangle at (250,180)-(321,201): text "%.0f bar"; shows P305.MaxBar; runs INTERN ASSIGN INPUTS.PresSelCalStbd[9]:=(FALSE); editable
rectangle at (360,180)-(431,201): text "%.0f bar"; shows P307.MaxBar; runs INTERN ASSIGN INPUTS.PresSelCalStbd[9]:=(FALSE); editable
rectangle at (470,180)-(541,201): text "%.0f bar"; shows P309.MaxBar; runs INTERN ASSIGN INPUTS.PresSelCalStbd[9]:=(FALSE); editable
rectangle at (580,180)-(651,201): text "%.0f bar"; shows P311.MaxBar; runs INTERN ASSIGN INPUTS.PresSelCalStbd[9]:=(FALSE); editable
rectangle at (470,395)-(541,416): text "%.1f %%"; shows PARAMS.stSE309Cfg.TgtLS_In; runs INTERN ASSIGN INPUTS.PresSelCalStbd[9]:=(FALSE); editable
rectangle at (470,495)-(541,516): text "%.1f %%"; shows PARAMS.stSE309Cfg.TgtLS_Out; runs INTERN ASSIGN INPUTS.PresSelCalStbd[9]:=(FALSE); editable
rounded rectangle at (470,335)-(541,371): text "ENABLE / MAX IN"; alarm colour if PARAMS.stSE309Cfg.LS_Limit_In; toggles PARAMS.stSE309Cfg.LS_Limit_In
rounded rectangle at (470,435)-(541,471): text "ENABLE / MAX OUT"; alarm colour if PARAMS.stSE309Cfg.LS_Limit_Out; toggles PARAMS.stSE309Cfg.LS_Limit_Out
rectangle at (40,295)-(111,316): text "%.1f %%"; shows PARAMS.stSE301Cfg.TgtLS_Slow; runs INTERN ASSIGN INPUTS.PresSelCalStbd[9]:=(FALSE); editable
rectangle at (40,280)-(111,296): text "LS Slow"
rectangle at (140,295)-(211,316): text "%.1f %%"; shows PARAMS.stSE303Cfg.TgtLS_Slow; runs INTERN ASSIGN INPUTS.PresSelCalStbd[9]:=(FALSE); editable
rectangle at (250,295)-(321,316): text "%.1f %%"; shows PARAMS.stSE305Cfg.TgtLS_Slow; runs INTERN ASSIGN INPUTS.PresSelCalStbd[9]:=(FALSE); editable
rectangle at (360,295)-(431,316): text "%.1f %%"; shows PARAMS.stSE307Cfg.TgtLS_Slow; runs INTERN ASSIGN INPUTS.PresSelCalStbd[9]:=(FALSE); editable
rectangle at (470,295)-(541,316): text "%.1f %%"; shows PARAMS.stSE309Cfg.TgtLS_Slow; runs INTERN ASSIGN INPUTS.PresSelCalStbd[9]:=(FALSE); editable
rectangle at (580,295)-(651,316): text "%.1f %%"; shows PARAMS.stSE311Cfg.TgtLS_Slow; runs INTERN ASSIGN INPUTS.PresSelCalStbd[9]:=(FALSE); editable
rectangle at (260,60)-(311,81): text "J5"
rectangle at (370,60)-(421,81): text "J4"
rectangle at (470,60)-(541,81): text "FORESTAY"
rectangle at (590,60)-(641,81): text "J2"
rectangle at (690,55)-(761,86): text "BACKSTAY / PORT"
rectangle at (790,55)-(861,86): text "BACKSTAY / STBD"
rectangle at (150,55)-(201,86): text "A3 / TACK"
rectangle at (50,55)-(101,86): text "FRO / TACK"
rectangle at (140,90)-(211,106): text "Time Max"
rectangle at (140,380)-(211,396): text "Max IN"
rectangle at (140,165)-(211,181): text "Pess. Max"
rectangle at (140,200)-(211,216): text "Press. Ease"
rectangle at (140,480)-(211,496): text "Max OUT"
rectangle at (140,125)-(211,141): text "Time Ease"
rectangle at (140,240)-(211,256): text "HP Pumps"
rectangle at (140,280)-(211,296): text "LS Slow"
rectangle at (250,90)-(321,106): text "Time Max"
rectangle at (250,380)-(321,396): text "Max IN"
rectangle at (250,165)-(321,181): text "Pess. Max"
rectangle at (250,200)-(321,216): text "Press. Ease"
rectangle at (250,480)-(321,496): text "Max OUT"
rectangle at (250,125)-(321,141): text "Time Ease"
rectangle at (250,240)-(321,256): text "HP Pumps"
rectangle at (250,280)-(321,296): text "LS Slow"
rectangle at (360,90)-(431,106): text "Time Max"
rectangle at (360,380)-(431,396): text "Max IN"
rectangle at (360,165)-(431,181): text "Pess. Max"
rectangle at (360,200)-(431,216): text "Press. Ease"
rectangle at (360,480)-(431,496): text "Max OUT"
rectangle at (360,125)-(431,141): text "Time Ease"
rectangle at (360,240)-(431,256): text "HP Pumps"
rectangle at (360,280)-(431,296): text "LS Slow"
rectangle at (470,90)-(541,106): text "Time Max"
rectangle at (470,380)-(541,396): text "Max IN"
rectangle at (470,165)-(541,181): text "Pess. Max"
rectangle at (470,200)-(541,216): text "Press. Ease"
rectangle at (470,480)-(541,496): text "Max OUT"
rectangle at (470,125)-(541,141): text "Time Ease"
rectangle at (470,240)-(541,256): text "HP Pumps"
rectangle at (470,280)-(541,296): text "LS Slow"
rectangle at (580,90)-(651,106): text "Time Max"
rectangle at (580,380)-(651,396): text "Max IN"
rectangle at (580,165)-(651,181): text "Pess. Max"
rectangle at (580,200)-(651,216): text "Press. Ease"
rectangle at (580,480)-(651,496): text "Max OUT"
rectangle at (580,125)-(651,141): text "Time Ease"
rectangle at (580,240)-(651,256): text "HP Pumps"
rectangle at (580,280)-(651,296): text "LS Slow"
rectangle at (745,90)-(816,106): text "Time Max"
rectangle at (745,380)-(816,396): text "Max IN"
rectangle at (695,165)-(766,181): text "Pess. P Max"
rectangle at (745,480)-(816,496): text "Max OUT"
rectangle at (745,125)-(816,141): text "Time Ease"
rectangle at (745,240)-(816,256): text "HP Pumps"
rounded rectangle at (905,55)-(1016,96): text "SAVE"; alarm colour if PARAMS.Save; toggles PARAMS.Save
22 more shapes without text or variables
*)

(* Visualisation VISU_CFG_CYLINDERS2
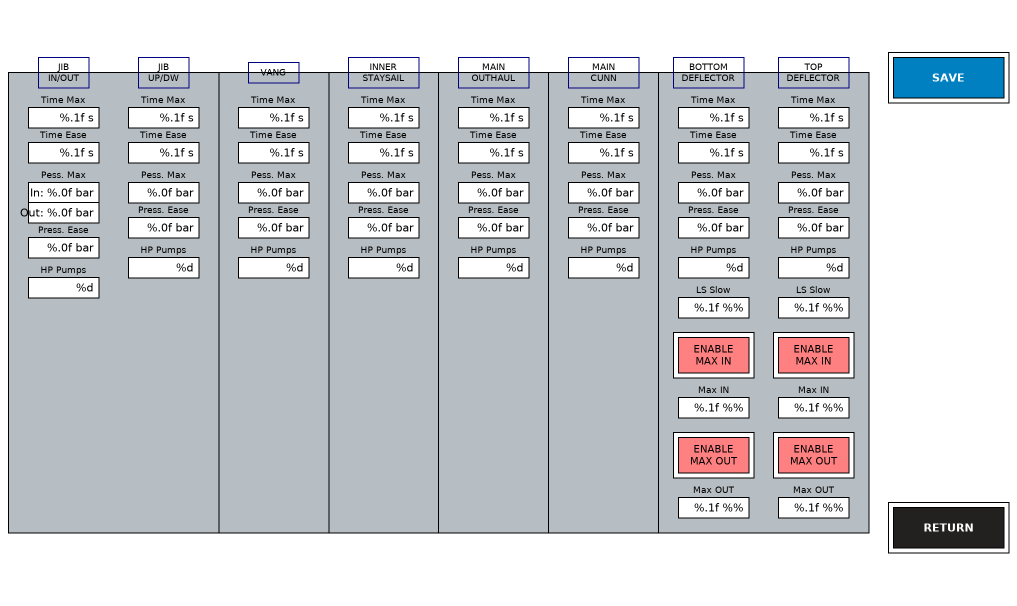
rectangle at (20,550)-(331,601): text "%s"; shows INPUTS.sVisuTime
rounded rectangle at (905,55)-(1016,96): text "SAVE"; alarm colour if PARAMS.Save; toggles PARAMS.Save
rounded rectangle at (905,505)-(1016,546): text "RETURN"; opens VISU_1_CYLINDERS2
rectangle at (730,550)-(896,601): text "SAVED!"; invisible if PARAMS.Saved
rectangle at (20,0)-(426,51): text "CFG: CYLINDERS 2"
rectangle at (40,90)-(111,106): text "Time Max"
rectangle at (40,165)-(111,181): text "Pess. Max"
rectangle at (40,235)-(111,256): text "%.0f bar"; shows PARAMS.stSE501Cfg.Ease; runs INTERN ASSIGN INPUTS.PresSelCalStbd[9]:=(FALSE); editable
rectangle at (40,220)-(111,236): text "Press. Ease"
rectangle at (40,140)-(111,161): text "%.1f s"; shows PARAMS.stSE501Cfg.TimeEase; runs INTERN ASSIGN INPUTS.PresSelCalStbd[9]:=(FALSE); editable
rectangle at (40,125)-(111,141): text "Time Ease"
rectangle at (40,275)-(111,296): text "%d"; shows PARAMS.stSE501Cfg.HP; runs INTERN ASSIGN INPUTS.PresSelCalStbd[9]:=(FALSE); editable 1..2
rectangle at (40,260)-(111,276): text "HP Pumps"
rectangle at (140,90)-(211,106): text "Time Max"
rectangle at (140,165)-(211,181): text "Pess. Max"
rectangle at (140,215)-(211,236): text "%.0f bar"; shows PARAMS.stSE503Cfg.Ease; runs INTERN ASSIGN INPUTS.PresSelCalStbd[9]:=(FALSE); editable
rectangle at (140,200)-(211,216): text "Press. Ease"
rectangle at (140,140)-(211,161): text "%.1f s"; shows PARAMS.stSE503Cfg.TimeEase; runs INTERN ASSIGN INPUTS.PresSelCalStbd[9]:=(FALSE); editable
rectangle at (140,125)-(211,141): text "Time Ease"
rectangle at (140,255)-(211,276): text "%d"; shows PARAMS.stSE503Cfg.HP; runs INTERN ASSIGN INPUTS.PresSelCalStbd[9]:=(FALSE); editable 1..2
rectangle at (140,240)-(211,256): text "HP Pumps"
rectangle at (250,215)-(321,236): text "%.0f bar"; shows PARAMS.stSE505Cfg.Ease; runs INTERN ASSIGN INPUTS.PresSelCalStbd[9]:=(FALSE); editable
rectangle at (250,140)-(321,161): text "%.1f s"; shows PARAMS.stSE505Cfg.TimeEase; runs INTERN ASSIGN INPUTS.PresSelCalStbd[9]:=(FALSE); editable
rectangle at (250,255)-(321,276): text "%d"; shows PARAMS.stSE505Cfg.HP; runs INTERN ASSIGN INPUTS.PresSelCalStbd[9]:=(FALSE); editable 1..2
rectangle at (690,395)-(761,416): text "%.1f %%"; shows PARAMS.stSE707Cfg.TgtLS_In; runs INTERN ASSIGN INPUTS.PresSelCalStbd[9]:=(FALSE); editable
rectangle at (690,380)-(761,396): text "Max IN"
rectangle at (360,215)-(431,236): text "%.0f bar"; shows PARAMS.stSE701Cfg.Ease; runs INTERN ASSIGN INPUTS.PresSelCalStbd[9]:=(FALSE); editable
rectangle at (690,495)-(761,516): text "%.1f %%"; shows PARAMS.stSE707Cfg.TgtLS_Out; runs INTERN ASSIGN INPUTS.PresSelCalStbd[9]:=(FALSE); editable
rectangle at (690,480)-(761,496): text "Max OUT"
rectangle at (360,140)-(431,161): text "%.1f s"; shows PARAMS.stSE701Cfg.TimeEase; runs INTERN ASSIGN INPUTS.PresSelCalStbd[9]:=(FALSE); editable
rectangle at (360,255)-(431,276): text "%d"; shows PARAMS.stSE701Cfg.HP; runs INTERN ASSIGN INPUTS.PresSelCalStbd[9]:=(FALSE); editable 1..2
rounded rectangle at (690,335)-(761,371): text "ENABLE / MAX IN"; alarm colour if PARAMS.stSE707Cfg.LS_Limit_In; toggles PARAMS.stSE707Cfg.LS_Limit_In
rounded rectangle at (690,435)-(761,471): text "ENABLE / MAX OUT"; alarm colour if PARAMS.stSE707Cfg.LS_Limit_Out; toggles PARAMS.stSE707Cfg.LS_Limit_Out
rectangle at (790,395)-(861,416): text "%.1f %%"; shows PARAMS.stSE709Cfg.TgtLS_In; runs INTERN ASSIGN INPUTS.PresSelCalStbd[9]:=(FALSE); editable
rectangle at (790,380)-(861,396): text "Max IN"
rectangle at (470,215)-(541,236): text "%.0f bar"; shows PARAMS.stSE703Cfg.Ease; runs INTERN ASSIGN INPUTS.PresSelCalStbd[9]:=(FALSE); editable
rectangle at (790,495)-(861,516): text "%.1f %%"; shows PARAMS.stSE709Cfg.TgtLS_Out; runs INTERN ASSIGN INPUTS.PresSelCalStbd[9]:=(FALSE); editable
rectangle at (790,480)-(861,496): text "Max OUT"
rectangle at (470,140)-(541,161): text "%.1f s"; shows PARAMS.stSE703Cfg.TimeEase; runs INTERN ASSIGN INPUTS.PresSelCalStbd[9]:=(FALSE); editable
rectangle at (470,255)-(541,276): text "%d"; shows PARAMS.stSE703Cfg.HP; runs INTERN ASSIGN INPUTS.PresSelCalStbd[9]:=(FALSE); editable 1..2
rounded rectangle at (790,335)-(861,371): text "ENABLE / MAX IN"; alarm colour if PARAMS.stSE709Cfg.LS_Limit_In; toggles PARAMS.stSE709Cfg.LS_Limit_In
rounded rectangle at (790,435)-(861,471): text "ENABLE / MAX OUT"; alarm colour if PARAMS.stSE709Cfg.LS_Limit_Out; toggles PARAMS.stSE709Cfg.LS_Limit_Out
rectangle at (580,215)-(651,236): text "%.0f bar"; shows PARAMS.stSE705Cfg.Ease; runs INTERN ASSIGN INPUTS.PresSelCalStbd[9]:=(FALSE); editable
rectangle at (580,140)-(651,161): text "%.1f s"; shows PARAMS.stSE705Cfg.TimeEase; runs INTERN ASSIGN INPUTS.PresSelCalStbd[9]:=(FALSE); editable
rectangle at (580,255)-(651,276): text "%d"; shows PARAMS.stSE705Cfg.HP; runs INTERN ASSIGN INPUTS.PresSelCalStbd[9]:=(FALSE); editable 1..2
rectangle at (690,215)-(761,236): text "%.0f bar"; shows PARAMS.stSE707Cfg.Ease; runs INTERN ASSIGN INPUTS.PresSelCalStbd[9]:=(FALSE); editable
rectangle at (690,140)-(761,161): text "%.1f s"; shows PARAMS.stSE707Cfg.TimeEase; runs INTERN ASSIGN INPUTS.PresSelCalStbd[9]:=(FALSE); editable
rectangle at (690,255)-(761,276): text "%d"; shows PARAMS.stSE707Cfg.HP; runs INTERN ASSIGN INPUTS.PresSelCalStbd[9]:=(FALSE); editable 1..2
rectangle at (790,215)-(861,236): text "%.0f bar"; shows PARAMS.stSE709Cfg.Ease; runs INTERN ASSIGN INPUTS.PresSelCalStbd[9]:=(FALSE); editable
rectangle at (790,140)-(861,161): text "%.1f s"; shows PARAMS.stSE709Cfg.TimeEase; runs INTERN ASSIGN INPUTS.PresSelCalStbd[9]:=(FALSE); editable
rectangle at (790,255)-(861,276): text "%d"; shows PARAMS.stSE709Cfg.HP; runs INTERN ASSIGN INPUTS.PresSelCalStbd[9]:=(FALSE); editable 1..2
rectangle at (40,180)-(111,201): text "In: %.0f bar"; shows P501.MaxBar; runs INTERN ASSIGN INPUTS.PresSelCalStbd[9]:=(FALSE); editable
rectangle at (140,180)-(211,201): text "%.0f bar"; shows P503.MaxBar; runs INTERN ASSIGN INPUTS.PresSelCalStbd[9]:=(FALSE); editable
rectangle at (250,180)-(321,201): text "%.0f bar"; shows P505.MaxBar; runs INTERN ASSIGN INPUTS.PresSelCalStbd[9]:=(FALSE); editable
rectangle at (360,180)-(431,201): text "%.0f bar"; shows P701.MaxBar; runs INTERN ASSIGN INPUTS.PresSelCalStbd[9]:=(FALSE); editable
rectangle at (470,180)-(541,201): text "%.0f bar"; shows P703.MaxBar; runs INTERN ASSIGN INPUTS.PresSelCalStbd[9]:=(FALSE); editable
rectangle at (580,180)-(651,201): text "%.0f bar"; shows P705.MaxBar; runs INTERN ASSIGN INPUTS.PresSelCalStbd[9]:=(FALSE); editable
rectangle at (690,180)-(761,201): text "%.0f bar"; shows P707.MaxBar; runs INTERN ASSIGN INPUTS.PresSelCalStbd[9]:=(FALSE); editable
rectangle at (790,180)-(861,201): text "%.0f bar"; shows P709.MaxBar; runs INTERN ASSIGN INPUTS.PresSelCalStbd[9]:=(FALSE); editable
rectangle at (40,105)-(111,126): text "%.1f s"; shows PARAMS.stSE501Cfg.TimeMax; runs INTERN ASSIGN INPUTS.PresSelCalStbd[9]:=(FALSE); editable
rectangle at (140,105)-(211,126): text "%.1f s"; shows PARAMS.stSE503Cfg.TimeMax; runs INTERN ASSIGN INPUTS.PresSelCalStbd[9]:=(FALSE); editable
rectangle at (250,105)-(321,126): text "%.1f s"; shows PARAMS.stSE505Cfg.TimeMax; runs INTERN ASSIGN INPUTS.PresSelCalStbd[9]:=(FALSE); editable
rectangle at (360,105)-(431,126): text "%.1f s"; shows PARAMS.stSE701Cfg.TimeMax; runs INTERN ASSIGN INPUTS.PresSelCalStbd[9]:=(FALSE); editable
rectangle at (470,105)-(541,126): text "%.1f s"; shows PARAMS.stSE703Cfg.TimeMax; runs INTERN ASSIGN INPUTS.PresSelCalStbd[9]:=(FALSE); editable
rectangle at (580,105)-(651,126): text "%.1f s"; shows PARAMS.stSE705Cfg.TimeMax; runs INTERN ASSIGN INPUTS.PresSelCalStbd[9]:=(FALSE); editable
rectangle at (690,105)-(761,126): text "%.1f s"; shows PARAMS.stSE707Cfg.TimeMax; runs INTERN ASSIGN INPUTS.PresSelCalStbd[9]:=(FALSE); editable
rectangle at (790,105)-(861,126): text "%.1f s"; shows PARAMS.stSE709Cfg.TimeMax; runs INTERN ASSIGN INPUTS.PresSelCalStbd[9]:=(FALSE); editable
rectangle at (40,200)-(111,221): text "Out: %.0f bar"; shows P507.MaxBar; runs INTERN ASSIGN INPUTS.PresSelCalStbd[9]:=(FALSE); editable
rectangle at (690,295)-(761,316): text "%.1f %%"; shows PARAMS.stSE707Cfg.TgtLS_Slow; runs INTERN ASSIGN INPUTS.PresSelCalStbd[9]:=(FALSE); editable
rectangle at (690,280)-(761,296): text "LS Slow"
rectangle at (790,295)-(861,316): text "%.1f %%"; shows PARAMS.stSE709Cfg.TgtLS_Slow; runs INTERN ASSIGN INPUTS.PresSelCalStbd[9]:=(FALSE); editable
rectangle at (790,280)-(861,296): text "LS Slow"
rectangle at (260,60)-(311,81): text "VANG"
rectangle at (50,55)-(101,86): text "JIB / IN/OUT"
rectangle at (150,55)-(201,86): text "JIB / UP/DW"
rectangle at (685,55)-(756,86): text "BOTTOM / DEFLECTOR"
rectangle at (790,55)-(861,86): text "TOP / DEFLECTOR"
rectangle at (360,55)-(431,86): text "INNER / STAYSAIL"
rectangle at (470,55)-(541,86): text "MAIN / OUTHAUL"
rectangle at (580,55)-(651,86): text "MAIN / CUNN"
rectangle at (250,90)-(321,106): text "Time Max"
rectangle at (250,165)-(321,181): text "Pess. Max"
rectangle at (250,200)-(321,216): text "Press. Ease"
rectangle at (250,125)-(321,141): text "Time Ease"
rectangle at (250,240)-(321,256): text "HP Pumps"
rectangle at (360,90)-(431,106): text "Time Max"
rectangle at (360,165)-(431,181): text "Pess. Max"
rectangle at (360,200)-(431,216): text "Press. Ease"
rectangle at (360,125)-(431,141): text "Time Ease"
rectangle at (360,240)-(431,256): text "HP Pumps"
rectangle at (470,90)-(541,106): text "Time Max"
rectangle at (470,165)-(541,181): text "Pess. Max"
rectangle at (470,200)-(541,216): text "Press. Ease"
rectangle at (470,125)-(541,141): text "Time Ease"
rectangle at (470,240)-(541,256): text "HP Pumps"
rectangle at (580,90)-(651,106): text "Time Max"
rectangle at (580,165)-(651,181): text "Pess. Max"
rectangle at (580,200)-(651,216): text "Press. Ease"
rectangle at (580,125)-(651,141): text "Time Ease"
rectangle at (580,240)-(651,256): text "HP Pumps"
rectangle at (690,90)-(761,106): text "Time Max"
rectangle at (690,165)-(761,181): text "Pess. Max"
rectangle at (690,200)-(761,216): text "Press. Ease"
rectangle at (690,125)-(761,141): text "Time Ease"
rectangle at (690,240)-(761,256): text "HP Pumps"
rectangle at (790,90)-(861,106): text "Time Max"
rectangle at (790,165)-(861,181): text "Pess. Max"
rectangle at (790,200)-(861,216): text "Press. Ease"
rectangle at (790,125)-(861,141): text "Time Ease"
rectangle at (790,240)-(861,256): text "HP Pumps"
12 more shapes without text or variables
*)

(* Visualisation VISU_CFG_ENGINE
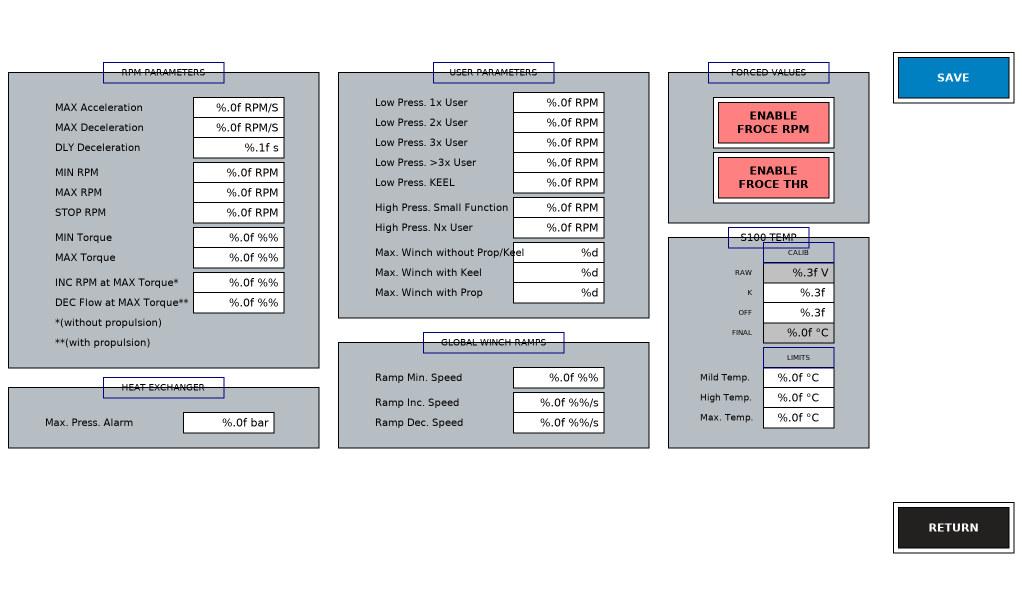
rectangle at (20,0)-(331,51): text "CFG: ENGINE"
rectangle at (20,550)-(331,601): text "%s"; shows INPUTS.sVisuTime
rounded rectangle at (905,55)-(1016,96): text "SAVE"; alarm colour if PARAMS.Save; toggles PARAMS.Save
rounded rectangle at (905,505)-(1016,546): text "RETURN"; opens VISU_1_ENGINE
rectangle at (110,60)-(231,81): text "RPM PARAMETERS"
rectangle at (520,195)-(611,216): text "%.0f RPM"; shows PARAMS.stEngineCfg.HP_SF_RPM; runs INTERN ASSIGN INPUTS.PresSelCalStbd[9]:=(FALSE); editable
rectangle at (520,90)-(611,111): text "%.0f RPM"; shows PARAMS.stEngineCfg.LP_1x_RPM; runs INTERN ASSIGN INPUTS.PresSelCalStbd[9]:=(FALSE); editable
rectangle at (520,110)-(611,131): text "%.0f RPM"; shows PARAMS.stEngineCfg.LP_2x_RPM; runs INTERN ASSIGN INPUTS.PresSelCalStbd[9]:=(FALSE); editable
rectangle at (380,90)-(511,111): text "Low Press. 1x User"; shows RECV_J1939.F004.DriverDemandTorque
rectangle at (520,130)-(611,151): text "%.0f RPM"; shows PARAMS.stEngineCfg.LP_3x_RPM; runs INTERN ASSIGN INPUTS.PresSelCalStbd[9]:=(FALSE); editable
rectangle at (520,150)-(611,171): text "%.0f RPM"; shows PARAMS.stEngineCfg.LP_Nx_RPM; runs INTERN ASSIGN INPUTS.PresSelCalStbd[9]:=(FALSE); editable
rectangle at (380,110)-(511,131): text "Low Press. 2x User"; shows RECV_J1939.F004.DriverDemandTorque
rectangle at (380,130)-(511,151): text "Low Press. 3x User"; shows RECV_J1939.F004.DriverDemandTorque
rectangle at (380,150)-(511,171): text "Low Press. >3x User"; shows RECV_J1939.F004.DriverDemandTorque
rectangle at (380,195)-(511,216): text "High Press. Small Function"; shows RECV_J1939.F004.DriverDemandTorque
rectangle at (200,95)-(291,116): text "%.0f RPM/S"; shows PARAMS.stEngineCfg.MaxInc_RPM; runs INTERN ASSIGN INPUTS.PresSelCalStbd[9]:=(FALSE); editable
rectangle at (200,115)-(291,136): text "%.0f RPM/S"; shows PARAMS.stEngineCfg.MaxDec_RPM; runs INTERN ASSIGN INPUTS.PresSelCalStbd[9]:=(FALSE); editable
rectangle at (200,160)-(291,181): text "%.0f RPM"; shows PARAMS.stEngineCfg.Min_RPM; runs INTERN ASSIGN INPUTS.PresSelCalStbd[9]:=(FALSE); editable 700..2600
rectangle at (200,180)-(291,201): text "%.0f RPM"; shows PARAMS.stEngineCfg.Max_RPM; runs INTERN ASSIGN INPUTS.PresSelCalStbd[9]:=(FALSE); editable 700..2600
rectangle at (60,95)-(191,116): text "MAX Acceleration"; shows RECV_J1939.F004.DriverDemandTorque
rectangle at (60,115)-(191,136): text "MAX Deceleration"; shows RECV_J1939.F004.DriverDemandTorque
rectangle at (60,160)-(191,181): text "MIN RPM"; shows RECV_J1939.F004.DriverDemandTorque
rectangle at (60,180)-(191,201): text "MAX RPM"; shows RECV_J1939.F004.DriverDemandTorque
rectangle at (440,60)-(561,81): text "USER PARAMETERS"
rectangle at (520,240)-(611,261): text "%d"; shows PARAMS.stEngineCfg.N_Winch_WOP; runs INTERN ASSIGN INPUTS.PresSelCalStbd[9]:=(FALSE); editable
rectangle at (380,240)-(511,261): text "Max. Winch without Prop/Keel"; shows RECV_J1939.F004.DriverDemandTorque
rectangle at (520,260)-(611,281): text "%d"; shows PARAMS.stEngineCfg.N_Winch_WK; runs INTERN ASSIGN INPUTS.PresSelCalStbd[9]:=(FALSE); editable
rectangle at (380,260)-(511,281): text "Max. Winch with Keel"; shows RECV_J1939.F004.DriverDemandTorque
rectangle at (200,225)-(291,246): text "%.0f %%"; shows PARAMS.stEngineCfg.Min_Torque; runs INTERN ASSIGN INPUTS.PresSelCalStbd[9]:=(FALSE); editable
rectangle at (200,245)-(291,266): text "%.0f %%"; shows PARAMS.stEngineCfg.Max_Torque; runs INTERN ASSIGN INPUTS.PresSelCalStbd[9]:=(FALSE); editable
rectangle at (60,225)-(191,246): text "MIN Torque"; shows RECV_J1939.F004.DriverDemandTorque
rectangle at (60,245)-(191,266): text "MAX Torque"; shows RECV_J1939.F004.DriverDemandTorque
rectangle at (200,270)-(291,291): text "%.0f %%"; shows PARAMS.stEngineCfg.Inc_RMP_Perc_WOP; runs INTERN ASSIGN INPUTS.PresSelCalStbd[9]:=(FALSE); editable
rectangle at (60,270)-(191,291): text "INC RPM at MAX Torque*"; shows RECV_J1939.F004.DriverDemandTorque
rectangle at (200,290)-(291,311): text "%.0f %%"; shows PARAMS.stEngineCfg.Dec_Flow_Perc_WP; runs INTERN ASSIGN INPUTS.PresSelCalStbd[9]:=(FALSE); editable
rectangle at (60,290)-(191,311): text "DEC Flow at MAX Torque**"; shows RECV_J1939.F004.DriverDemandTorque
rectangle at (110,375)-(231,396): text "HEAT EXCHANGER"
rectangle at (190,410)-(281,431): text "%.0f bar"; shows PARAMS.stEngineCfg.Max_HeatExch_P; runs INTERN ASSIGN INPUTS.PresSelCalStbd[9]:=(FALSE); editable
rectangle at (50,410)-(181,431): text "Max. Press. Alarm"; shows RECV_J1939.F004.DriverDemandTorque
rectangle at (60,310)-(191,331): text "*(without propulsion)"; shows RECV_J1939.F004.DriverDemandTorque
rectangle at (60,330)-(191,351): text "**(with propulsion)"; shows RECV_J1939.F004.DriverDemandTorque
rectangle at (200,135)-(291,156): text "%.1f s"; shows PARAMS.stEngineCfg.DlyDec_sec; runs INTERN ASSIGN INPUTS.PresSelCalStbd[9]:=(FALSE); editable
rectangle at (60,135)-(191,156): text "DLY Deceleration"; shows RECV_J1939.F004.DriverDemandTorque
rectangle at (505,550)-(671,601): text "SAVED!"; invisible if PARAMS.Saved
rectangle at (520,170)-(611,191): text "%.0f RPM"; shows PARAMS.stEngineCfg.LP_CK_RPM; runs INTERN ASSIGN INPUTS.PresSelCalStbd[9]:=(FALSE); editable
rectangle at (380,170)-(511,191): text "Low Press. KEEL"; shows RECV_J1939.F004.DriverDemandTorque
rectangle at (520,365)-(611,386): text "%.0f %%"; shows PARAMS.stWRAMPCfg.Spd_Min; runs INTERN ASSIGN INPUTS.PresSelCalStbd[9]:=(FALSE); editable
rectangle at (520,390)-(611,411): text "%.0f %%/s"; shows PARAMS.stWRAMPCfg.Spd_Inc; runs INTERN ASSIGN INPUTS.PresSelCalStbd[9]:=(FALSE); editable
rectangle at (520,410)-(611,431): text "%.0f %%/s"; shows PARAMS.stWRAMPCfg.Spd_Dec; runs INTERN ASSIGN INPUTS.PresSelCalStbd[9]:=(FALSE); editable
rectangle at (430,330)-(571,351): text "GLOBAL WINCH RAMPS"
rectangle at (380,365)-(511,386): text "Ramp Min. Speed"; shows RECV_J1939.F004.DriverDemandTorque
rectangle at (380,390)-(511,411): text "Ramp Inc. Speed"; shows RECV_J1939.F004.DriverDemandTorque
rectangle at (380,410)-(511,431): text "Ramp Dec. Speed"; shows RECV_J1939.F004.DriverDemandTorque
rectangle at (200,200)-(291,221): text "%.0f RPM"; shows PARAMS.stEngineCfg.STOP_RPM; runs INTERN ASSIGN INPUTS.PresSelCalStbd[9]:=(FALSE); editable 700..2600
rectangle at (60,200)-(191,221): text "STOP RPM"; shows RECV_J1939.F004.DriverDemandTorque
rectangle at (715,60)-(836,81): text "FORCED VALUES"
rounded rectangle at (725,100)-(836,141): text "ENABLE / FROCE RPM"; alarm colour if PARAMS.stEngineCfg.EnForceRPM; toggles PARAMS.stEngineCfg.EnForceRPM
rounded rectangle at (725,155)-(836,196): text "ENABLE / FROCE THR"; alarm colour if PARAMS.stEngineCfg.EnForceTHR; toggles PARAMS.stEngineCfg.EnForceTHR
rectangle at (520,280)-(611,301): text "%d"; shows PARAMS.stEngineCfg.N_Winch_WP; runs INTERN ASSIGN INPUTS.PresSelCalStbd[9]:=(FALSE); editable
rectangle at (380,280)-(511,301): text "Max. Winch with Prop"; shows RECV_J1939.F004.DriverDemandTorque
rectangle at (520,215)-(611,236): text "%.0f RPM"; shows PARAMS.stEngineCfg.HP_Nx_RPM; runs INTERN ASSIGN INPUTS.PresSelCalStbd[9]:=(FALSE); editable
rectangle at (380,215)-(511,236): text "High Press. Nx User"; shows RECV_J1939.F004.DriverDemandTorque
rectangle at (705,365)-(771,386): text "Mild Temp."
rectangle at (770,365)-(841,386): text "%.0f °C"; shows S100.LowDeg; runs INTERN ASSIGN INPUTS.PresSelCalStbd[9]:=(FALSE); editable
rectangle at (705,385)-(771,406): text "High Temp."
rectangle at (770,385)-(841,406): text "%.0f °C"; shows S100.HigDeg; runs INTERN ASSIGN INPUTS.PresSelCalStbd[9]:=(FALSE); editable
rectangle at (705,405)-(771,426): text "Max. Temp."
rectangle at (770,405)-(841,426): text "%.0f °C"; shows S100.MaxDeg; runs INTERN ASSIGN INPUTS.PresSelCalStbd[9]:=(FALSE); editable
rectangle at (710,260)-(761,281): text "RAW"
rectangle at (710,320)-(761,341): text "FINAL"
rectangle at (710,280)-(761,301): text "K"
rectangle at (710,300)-(761,321): text "OFF"
rectangle at (735,225)-(816,246): text "S100 TEMP"
rectangle at (770,320)-(841,341): text "%.0f °C"; shows S100.Deg
rectangle at (770,280)-(841,301): text "%.3f"; shows S100.Cal_K; runs INTERN ASSIGN INPUTS.PresSelCalStbd[9]:=(FALSE); editable
rectangle at (770,260)-(841,281): text "%.3f V"; shows S100.Raw; alarm colour if S100.Err; runs INTERN ASSIGN INPUTS.PresSelCalStbd[9]:=(FALSE)
rectangle at (770,300)-(841,321): text "%.3f"; shows S100.Cal_Off; runs INTERN ASSIGN INPUTS.PresSelCalStbd[9]:=(FALSE); editable
rectangle at (770,240)-(841,261): text "CALIB"
rectangle at (770,345)-(841,366): text "LIMITS"
10 more shapes without text or variables
*)

